(* CODESYS project RoofTrussLibrary.library
   Author: Sawtooth Engineers
   Version: 0.1.0.0
   Description: Containes components and equipment modules for base components of a roof truss core system.
   Title: RoofTrussLibrary
   DefaultNamespace: RTL
   Placeholder: RoofTrussLibrary
   Company: Sawtooth Robotics

Project tree, tasks and I/O mapping:
  libraries: Recipe Management, * (System); SPT Base Types, * (Beckhoff Automation LLC); SPT Components, * (Beckhoff Automation LLC); SPT Event Logger, * (Beckhoff Automation LLC); SPT Motion Control, * (Beckhoff Automation LLC); Tc2_NcDrive, * (Beckhoff Automation GmbH); Tc2_Standard, * (Beckhoff Automation GmbH); Tc2_System, * (Beckhoff Automation GmbH); Tc2_TcpIp, * (Beckhoff Automation GmbH); Tc2_Utilities, * (Beckhoff Automation GmbH); Tc3_Database, * (Beckhoff Automation GmbH); Tc3_EventLogger, * (Beckhoff Automation GmbH); Tc3_JsonXml, * (Beckhoff Automation GmbH); Tc3_PackML_V2, * (Beckhoff Automation GmbH)
  DUTs/
    DB_Logging/
      data type ST_EquipmentModuleLog
    MessageBoxes/
      data type ST_Active_MessageBoxes
      data type ST_MessageBox_Button
      data type ST_MessageBox_Buttons
      data type ST_MessageBox_Data
      data type ST_MessageBox_Messages
      data type ST_MessageBox_Response
    Motion/
      data type E_SpeedOptions
      data type ST_HomingParams
      data type ST_MoveStates
    Recipe/
      data type E_CommandName
      data type E_RamState
      data type ST_AssemblyData
      data type ST_AssemblyEnd
      data type ST_AssemblyStart
      data type ST_AxisRecipe
      data type ST_Board
      data type ST_BoardData
      data type ST_BoardInfo
      data type ST_CSV
      data type ST_CSV_Detail
      data type ST_CSV_Generic
      data type ST_CSV_Line
      data type ST_CSV_Step
      data type ST_Detail_Descriptions
      data type ST_IndexConveyor
      data type ST_KeyValue
      data type ST_PickPlace
      data type ST_PickPlaceDetail
      data type ST_PlateInfo
      data type ST_Plates
      data type ST_PositionInfo
      data type ST_PressRecipe
      data type ST_TrussInfo
    WaitSync/
      data type E_EM_Index
      data type E_WaitSync
      data type ST_WaitSyncManager
    data type E_AssemblyPickState
    data type E_BoardData_Positions
    data type E_CarriageStates
    data type E_Double_Pick_States
    data type E_GrabState
    data type E_Infeed_States
    data type E_Location_IDs
    data type E_MBI_States
    data type E_MoveCarriageState
    data type E_Outfeed_Conveyor_State
    data type E_Outfeed_Conveyor_SubState
    data type E_Press_States
    data type E_ReleaseState
    data type ST_BEPointDefinitions
    data type ST_BoardLengthTest
    data type ST_BoardLengthTestData
    data type ST_ConveyorData
    data type ST_DualChannel_HMIStatus
    data type ST_MGBDoor_HMIStatus
    data type ST_MotorControls_NonStandard
    data type ST_OutfeedConveyorStatus
    data type ST_PackML_Control
    data type ST_PackML_Control_Simplified
    data type ST_RecoveryBoardList
    data type ST_SysConfig
  GVLs/
    global variables Global
  Machine/
    Components/
      BasicSlaveAxis_SOE/
        DUTs/
          HMI/
            data type ST_MyComponent_Command_1
            data type ST_MyComponent_Config_1
            data type ST_MyComponent_HMI_1
            data type ST_MyComponent_Status_1
        Interfaces/
        function block FB_Component_BasicSlaveAxis_SoE [ST]: CyclicLogic, Reset
      Button/
        DUTs/
        Interfaces/
        function block FB_Component_Button [ST]: CyclicLogic, CreateEvents, Initialize, Monitoring, Button_Pressed
      ComponentBase_SR/
        Interfaces/
          interface I_ComponentBase_SR
        function block FB_ComponentBase_SR [ST]: ClearAlarms, RaiseAlarm2Args, Reset
      ControlPendant/
        DUTs/
        Interfaces/
        function block FB_ControlPendant [ST]: CyclicLogic, CreateEvents, Initialize, Monitoring, Mode_Auto, Mode_Idle, Mode_Manual_1, Mode_Manual_2
        function block FB_ControlPendant_Outfeed [ST]: CyclicLogic, CreateEvents, Initialize, Monitoring
      Conveyor/
        DUTs/
          HMI/
        Interfaces/
        function block FB_Conveyor [ST]: CyclicLogic, AlarmRaiseBasic, CreateEvents, Monitoring, SimHoming, ParentResponseDefinitions
      DoubleSolenoidRetractFeedback/
        DUT/
        Interfaces/
        function block FB_DoubleSolenoidRetractFeedback [ST]: Feedback, HardwareInit, RetractedInput
      DualChannelIndicator/
        function block FB_DualChannelMonitor [ST]: CyclicLogic, CreateEvents, Initialize, BothChannelsOK
      Indicator/
        DUTs/
          HMI/
            data type ST_Indicator_Command
            data type ST_Indicator_Config
            data type ST_Indicator_HMI
            data type ST_Indicator_Status
        Interfaces/
          interface I_Indicator: Flash, TurnOff, TurnOn
        function block FB_Component_Indicator [ST]: CyclicLogic, CreateEvents, Flash, Initialize, Monitoring, Reset, TurnOff, TurnOn, Flashing, Off, OffTime, On, OnTime
      IRC5/
        DUTs/
          HMI/
            data type ST_IRC5_Command
            data type ST_IRC5_Config
            data type ST_IRC5_HMI
            data type ST_IRC5_Status
          data type ST_IRC5_Input
          data type ST_IRC5_IO
          data type ST_IRC5_Output
        Interfaces/
          interface I_IRC5
        function block FB_Component_IRC5 [ST]: CyclicLogic, Abort, CreateEvents, EStopReset, Initialize, Monitoring, SignalMapping, Start, Stop, EStopped, InAuto, ParentResponseDefinitions
      MGB_Door/
        DUTs/
          HMI/
        Interfaces/
        function block FB_Component_MGB_Door [ST]: CyclicLogic, HMI_Status, Initialize, AutoStop_CH_OK, Estop_CH_OK, SafetyReset
      Preplate_Rack/
        DUTs/
          HMI/
          data type E_RackState
          data type linked_racks_typ
          data type RackStateMachine
          data type RackStatus
        Interfaces/
        function block FB_Component_Preplate_Rack [ST]: CyclicLogic, Block, Disable, Initialize, IsAvailable, RackLogic, Blocked, InAuto, LinkBlocked
      Robot/
        DUTs/
          data type ST_Robot_Handshake_Input
          data type ST_Robot_Handshake_IO
          data type ST_Robot_Handshake_Output
        Interfaces/
        function block FB_Component_Robot [ST]: CyclicLogic, Clear_DataToSend, CreateEvents, HandshakeSignalMapping, Initialize, Monitoring, PackRecipeData, OtherInputs, OtherOutputs
      Safety/
        DUTs/
          HMI/
        Interfaces/
        function block FB_Component_Safety [ST]: CyclicLogic, CreateEvents, HMI_Indicators, HMI_Status_Estops, HMI_Status_LightCurtains, HMI_Status_Preplate, Initialize, Monitoring, PauseInputs, ResumeInputs, AutostopOK, OutfeedAutostopOK, ParentResponseDefinitions, SafetyOK, SystemState
      StackLight/
        DUTs/
          HMI/
        Interfaces/
          interface I_StackLight: SystemErrorPresent
        function block FB_Component_Stacklight [ST]: CyclicLogic, CreateEvents, Initialize, Monitoring, SystemErrorPresent, SystemState
      StackLight_MBI/
        Interfaces/
          interface I_StackLight_1: MyInput, MyOutput
        function block FB_Component_Stacklight_MBI [ST]: CyclicLogic, CreateEvents, Initialize, Monitoring, MyOutput, SystemErrorPresent
      Template_MyComponent/
        DUTs/
          HMI/
            data type ST_MyComponent_Command
            data type ST_MyComponent_Config
            data type ST_MyComponent_HMI
            data type ST_MyComponent_Status
        Interfaces/
          interface I_MyComponent: SystemErrorPresent, SystemState
        function block FB_Component_MyComponent [ST]: CyclicLogic, CreateEvents, Initialize, Monitoring, MyInput, MyOutput
      VFD/
        DUTs/
          HMI/
        Interfaces/
          interface I_VFD: Jog, Stop
        function block FB_Component_ABB_VFD_EC [ST]: CyclicLogic, Extended, Retracted, Jog, Reset, Stop
        function block FB_Component_ABB_VFD_EIP [ST]: CyclicLogic, Disable, Enable, Initialize, Jog, Monitoring, Reset, Stop, AtSpeed, CommandedVel, Enabled, Faulted, FaultReset, Frequency, FwdActive, JogFwd, JogRvs, ReferenceVel, RvsActive, State, Warning
    EquipmentModules/
      EquipmentModule_SR/
        Interfaces/
          interface I_CommandStepParser: AssemblyEndParse, AssemblyStartParse, BoardInfoParse, BoardParse, NailPlateParse, TrussInfoParse
          interface I_CommandSteps: AssemblyEnd, AssemblyStart, Board, BoardInfo, NailPlate, TrussInfo
          interface I_EquipmentModule_SR: EquipmentModuleID, InSimulation, SafetyOK, SimulationOff, SimulationOn
          interface I_MachineComms: Step, WaitSync
        function block FB_EquipmentModule_SR [ST]: AssemblyEndParse, AssemblyStartParse, BoardInfoParse, BoardParse, IndexConveyorParse, NailPlateParse, PickPlaceParse, TrussInfoParse, CyclicLogic, CyclicLogicSimulation, Step, AssignMessageBox, ComponentMonitor, EM_BufferLogging, HMIControl, LengthFormatString, MotorResetAndEnable, MotorsHome, MotorsInit, MotorsInitAlignGearIn, RaiseAlarm2Args, RaiseMessageBox, RegisterSubmodules, ResetMessageBox, ResetOnResume, RestartStateCheck, SimHoming, SubModuleMonitor, TorqueHoming, TorqueHoming_old, WaitSync_Handler, WaitSync_ReadWrite, WaitSyncCheck, Holding, Resetting, Starting, Suspending, Unholding, Unsuspending, Execute, Idle, Suspended, CurrentStep, EquipmentModuleID, ForceHold, ParentResponseDefinitions, RecoverBoardNum, SafetyOK, TaskState, ClearAlarms, ResetComponents, InSimulation, SimulationOff, SimulationOn
      Functional Layer/
        function block FB_Carriage [ST]: CyclicLogic, Starting, Unholding, Unsuspending, CreateEvents, GrabBoard, HMIControl, Initialize, Monitoring, MotorsInit, MoveIdleOnStarting, ReleaseBoard, SetSpeeds, TestLengthPosCompare, ZPrepMove, ActuatorsClosed, ActuatorsOpen, AxisRef, BoardHeight, BoardSecured, ClearOfBoards, ClearOfCarriages, CloseActuatorsRequest, HoldingBoard, IdlePos, IgnoreSensors, MasterAxis, MoveClearActive, MovementRequested, MoveState, MoveSubState, OpenActuatorsRequest, OverrideSensors, PressPermissions, Request_WS, Response_WS, TargetPos
        function block FB_Handoff [ST]: CyclicLogic, GrabBoard, HMIControl, Initialize, ReleaseBoard, ClampsClosed, ClampsOpen, DisableClamp1, DisableClamp2, HoldingBoard, Location, Request_WS, Response_WS
        function block FB_Infeed [ST]: CyclicLogic, Aborting, Holding, Starting, Stopping, Suspending, ExecuteStep, Execute, Auto, ClearInfeed, CreateEvents, HMIControl, Initialize, Monitoring, ParseBoardData, RoughLengthCheck, SimpAuto, SuperSimpAuto, ActiveInfeedMoving, BoardDataToPass, BoardDropped, BoardReadyForCarriage, Carriage1LengthTesting, Carriage1ResetInfeed_Request, Carriage2_DoublePickCancel_Request, Carriage2ResetInfeed_Request, CarriageClearOfBoardPresentSensor, IgnoreDoublePick, InfeedToInfeedReady, InfeedToInfeedRequest, LineNumber, MoveClearActive, ParentState, ReadyForBoard, Sim_InfeedClear, TestExecute
        function block FB_MBI [ST]: CyclicLogic, Aborting, Holding, Starting, Stopping, Suspending, Unholding, Unsuspending, Aborted, Execute, Held, Idle, Stopped, Suspended, Auto, CreateEvents, HMIControl, Initialize, ManualMode_Forward, ManualMode_Reverse, Monitoring, Production, BoardDropped, LineNumber, MainSafetyOK, ParentState, ReadyForBoard, TestExecute
        function block FB_Outfeed_Jig [ST]: CyclicLogic, Suspending, Unsuspending, ExecuteStep, RunIndexConveyor, RunPickPlace, RunTrussInfo, Aborted, Execute, Held, Idle, Stopped, Suspended, ComponentMonitor, CreateEvents, HMIControl, IndexFull, IndexHalf, Initialize, Monitoring, MotorsInit, NewTrussInfo, OutfeedConveyorLogic, PopulateBoardToArray, AutostopOK, MainSafetyOK, MaxConveyorCount, OutfeedAutostopOK, OutfeedConveyorStatus, ParentState, PickPlace_Done_ENUM, PickPlace_Ready_ENUM
        function block FB_Preplate [ST]: CyclicLogic, Execute, HMIControl, Initialize, InAuto
        function block FB_Press [ST]: CyclicLogic, Aborting, Clearing, Holding, Starting, Stopping, Suspending, Unholding, Unsuspending, AssemblyEnd, AssemblyStart, ExecuteDetail, ExecuteStep, Execute, DoublePickNailPlatePosCheck, HMIControl, Initialize, MotorsInit, PressLogic, BoardDataToPass, DoublePickData_Ready, DoublePickData_Sent, DoublePickDataToPass, NailplateCountData_Ready, NailplateCountData_Sent, NailplateDataToPass, PressRobotPermissionToEnter
        function block FB_Robot [ST]: CyclicLogic, CyclicLogicSimulation, Aborting, Clearing, Completing, Holding, Resetting, Starting, Stopping, Suspending, Unholding, Unsuspending, NailPlate, Execute, ExtractNumFromString, HMIControl, Initialize, WaitSync_Robot, DryRun, OtherInputs, OtherOutputs, SubModuleMonitor
        function block FB_Robot_Outfeed [ST]: CyclicLogic, CyclicLogicSimulation, ExecuteDetail, ExecuteDetail_SIM, ExecuteStep, HMIControl, Initialize, UI_MessageBox, PickPlaceDataToPass
        function block FB_Robot_PrePlate [ST]: CyclicLogic, CyclicLogicSimulation, ExecuteDetail, ExecuteDetail_SIM, ExecuteStep, HMIControl, Initialize, UI_MessageBox
        function block FB_Robot_Press [ST]: CyclicLogic, CyclicLogicSimulation, ExecuteDetail, ExecuteDetail_SIM, ExecuteStep, HMIControl, Initialize, UI_MessageBox
      Info Layer/
        function block _FB_EquipmentModule_Info [ST]: CyclicLogic, Aborting, FindBoardForRecovery, Task
      SamComm/
        DUTs/
          HMI/
          data type E_ContentType
          data type E_MessageCategory
          data type E_MessageStatus
          data type E_SAMCommStateMachine
          data type E_TaskState
          data type ST_Alert
          data type ST_Message
          data type ST_Messages
          data type ST_PLC
          data type ST_RFT
          data type ST_Status
          data type ST_Task
          data type ST_Task_Info
          data type ST_TaskREF
          data type ST_TaskStatus
        Helper POUs/
          function block FB_FrameFifo [ST]: AddTail, Clear, RemoveHead, Send
          function block FB_LogFifo [ST]: Clear, Error, Message, Remove
        function block FB_ClientConnection [ST]
        function block FB_SamComm [ST]: CyclicLogic, CheckForRFT, CheckForStatusUpdate, ComposeRequestForInfo, ComposeRFT, ComposeStatus, ExtractMetaData, GenUUID, InfeedLineNumberCheck, IsIdleTask, ParseCSVData, ProcessReceivedMessage, STRING_TO_E_CommandName, Application, CreateEvents, Initialize, RaiseAlarm2Args, OutfeedConveyorStatus_Jig2, OutfeedConveyorStatus_Jig3, Tasks
      Templates/
    Events/
      AMDTruss.tmc
    FunctionBlocks/
      Occupy Press Street/
        data type E_GateKeeperState
        data type ST_MediatorInterface
      PulseGenerator/
        Interfaces/
          interface I_PulseGenerator: OffTime, OnTime, PulseOutput
        function block FB_PulseGenerator [ST]: CyclicLogic, OffTime, OnTime, PulseOutput
    HMI Connections/
      function block FB_ControlSource_HMI [ST]: CyclicLogic, Control, ModeChanged, StateChanged, ForceHoldRequested, Initialize, Registered
      function block FB_ControlSource_HMI_Machine [ST]: CyclicLogic
      function block FB_ControlSource_MBI [ST]: CyclicLogic, Control, ModeChanged, StateChanged, Initialize, Registered
  00000000-0000-0000-0000-000000000000|Machine\Events\AMDTruss.tmc
  Project Information/
    function F_GetCompany [ST]
    function F_GetTitle [ST]
    function F_GetVersion [ST]
  Version/
    global variables Global_Version
  text list GlobalTextList
*)

// DUTs/DB_Logging/ST_EquipmentModuleLog
TYPE
    ST_EquipmentModuleLog : STRUCT
        Timestamp   : DT;
        ModuleName  : STRING(32);
        PackMLState : STRING(32);
        Message     : STRING(255);
    END_STRUCT
END_TYPE

// DUTs/MessageBoxes/ST_Active_MessageBoxes
TYPE
    ST_Active_MessageBoxes : STRUCT
        SelectedTabIndex          : USINT;
        MessageBox_Data           : ARRAY[1..30] OF ST_MessageBox_Data;
        Displayed_MessageBox_Data : ST_MessageBox_Data;
        ErrorSolution             : USINT;
        ErrorAcknowledge          : BOOL;
    END_STRUCT
END_TYPE

// DUTs/MessageBoxes/ST_MessageBox_Button
TYPE
    ST_MessageBox_Button : STRUCT
        Text    : STRING;
        Visible : BOOL;
    END_STRUCT
END_TYPE

// DUTs/MessageBoxes/ST_MessageBox_Buttons
TYPE
    ST_MessageBox_Buttons : STRUCT
        Button1 : ST_MessageBox_Button;
        Button2 : ST_MessageBox_Button;
        Button3 : ST_MessageBox_Button;
        Button4 : ST_MessageBox_Button;
        Button5 : ST_MessageBox_Button;
    END_STRUCT
END_TYPE

// DUTs/MessageBoxes/ST_MessageBox_Data
TYPE
    ST_MessageBox_Data : STRUCT
        Equipment_Module        : E_EM_Index;
        Equipment_Module_String : STRING;
        TimeStamp               : STRING;
        Header                  : STRING[80];
        Icon                    : USINT;
        Severity                : TcEventSeverity;
        Messages                : ST_MessageBox_Messages;
        Buttons                 : ST_MessageBox_Buttons;
        ErrorPresent            : BOOL;
        ErrorNumber             : UINT;
    END_STRUCT
END_TYPE

// DUTs/MessageBoxes/ST_MessageBox_Messages
TYPE
    ST_MessageBox_Messages : STRUCT
        Message1 : STRING[80];
        Message2 : STRING[80];
        Message3 : STRING[80];
        Message4 : STRING[80];
        Message5 : STRING[80];
        Message6 : STRING[80];
        Message7 : STRING[80];
    END_STRUCT
END_TYPE

// DUTs/MessageBoxes/ST_MessageBox_Response
TYPE
    ST_MessageBox_Response : STRUCT
        ErrorRaised      : BOOL;
        ErrorAcknowledge : BOOL;
        ErrorSolution    : USINT;
    END_STRUCT
END_TYPE

// DUTs/Motion/E_SpeedOptions
{attribute 'qualified_only'}
{attribute 'strict'}
{attribute 'to_string'}
TYPE
    E_SpeedOptions : (
        AUTO        := 1,
        MANUAL      := 2,
        MAINTENANCE := 3,
        TESTING1    := 4,
        TESTING2    := 5,
        TESTING3    := 6,
        TESTING4    := 7,
        TESTING5    := 8
    );
END_TYPE

// DUTs/Motion/ST_HomingParams
TYPE
    ST_HomingParams : STRUCT
        ReadParams               : SPT_Motion_Control.MC_ReadParameter;
        WriteNegLim              : SPT_Motion_Control.MC_WriteBoolParameter;
        WritePosLim              : SPT_Motion_Control.MC_WriteBoolParameter;
        AxisParams               : SPT_Motion_Control.MC_AxisParameter;
        SetPositionHomingRoutine : FB_HomeRoutine_SetPosition;
        TorqueControl            : SPT_Motion_Control.MC_TorqueControl;
        TorqueControlParams      : SPT_Motion_Control.ST_TorqueControlOptions;
        HardStopHomingRoutine    : FB_HomeRoutine_HardStop;
        HardStopHomingParams     : ST_StepBlockLagBasedParameters;
        SetPositionOffset        : SPT_Motion_Control.FB_CoEAX8000SetPositionOffset;
        HomingTON                : TON;
        Execute_WriteLimit       : BOOL;
        EnablePosLim             : BOOL;
        EnableNegLim             : BOOL;
        HomingState              : DINT;
        HomePosMax               : LREAL;
        HomePosMin               : LREAL;
    END_STRUCT
END_TYPE

// DUTs/Motion/ST_MoveStates
TYPE
    ST_MoveStates : STRUCT
        Idle    : UDINT;
        Pick    : UDINT;
        Hold    : UDINT;
        Clear   : UDINT;
        Drop    : UDINT;
        Grab    : UDINT;
        Release : UDINT;
    END_STRUCT
END_TYPE

// DUTs/Recipe/E_CommandName
{attribute 'qualified_only'}
{attribute 'strict'}
{attribute 'to_string'}
TYPE
    E_CommandName : (
        Unknown       := 0,
        AssemblyStart := 1,
        TrussInfo     := 2,
        PuckMove      := 3,
        PickPlace     := 4,
        IndexConveyor := 5,
        ManualBoard   := 6,
        BoardInfo     := 7,
        Board         := 8,
        NailPlate     := 9,
        ManualPlate   := 10,
        AssemblyEnd   := 11
    );
END_TYPE

// DUTs/Recipe/E_RamState
{attribute 'qualified_only'}
{attribute 'strict'}
{attribute 'to_string'}
TYPE
    E_RamState : (
        rsINIT,
        rsIDLE,
        rsFULL_RETRACT,
        rsFULL_EXTEND,
        rsSEND_TO_POSITION,
        rsEXTEND_TO_BACKER,
        rsEXTEND_TO_CLOSED_PREP,
        rsEXTEND_TO_CLOSED,
        rsFAILED_TO_CYCLE,
        rsEXTENDING_TO_PRESSURE,
        rsEXTEND_TO_PRESSURE,
        rsRETRACT_FOR_INDEX,
        rsUNDEFINED,
        rsERROR
    );
END_TYPE

// DUTs/Recipe/ST_AssemblyData
TYPE
    ST_AssemblyData : STRUCT
        Boards : ARRAY[1..MAX_NUMBER_OF_BOARDS] OF ST_BoardData;
    END_STRUCT
END_TYPE

// DUTs/Recipe/ST_AssemblyEnd
TYPE
    ST_AssemblyEnd : STRUCT
        SeqID : UDINT;
    END_STRUCT
END_TYPE

// DUTs/Recipe/ST_AssemblyStart
TYPE
    ST_AssemblyStart : STRUCT
        ComponentID : T_MaxString;
    END_STRUCT
END_TYPE

// DUTs/Recipe/ST_AxisRecipe
TYPE
    ST_AxisRecipe : STRUCT
        Velocity     : LREAL := 150;
        Acceleration : LREAL := 300;
        Torque       : LREAL := 100;
    END_STRUCT
END_TYPE

// DUTs/Recipe/ST_Board
TYPE
    ST_Board : STRUCT
        BoardID                 : STRING;
        BoardWidth              : REAL;
        BoardHeight             : REAL;
        BoardLength             : REAL;
        BoardNumber             : INT;
        LeadingEdgeBevelOffset  : REAL;
        TrailingEdgeBevelOffset : REAL;
    END_STRUCT
END_TYPE

// DUTs/Recipe/ST_BoardData
TYPE
    ST_BoardData : STRUCT
        BoardID                       : STRING;
        BoardWidth                    : REAL;
        BoardHeight                   : REAL;
        BoardLength                   : REAL;
        BoardLength_Measured          : BOOL;
        BoardNumber                   : INT;
        Plates_Total                  : UDINT;
        Plates_Placed                 : UDINT;
        TotalPlateCount_Data_Received : BOOL;
        LeadingEdgeBevelOffset        : REAL;
        TrailingEdgeBevelOffset       : REAL;
        PickOffset                    : REAL;
        DoublePickNeeded              : BOOL;
        DoublePickVerified            : BOOL;
        DoublePicked                  : BOOL;
        IgnoreSensors                 : BOOL;
        FrontEdgePos                  : REAL;
        BackEdgePos                   : REAL;
        LocationStr                   : STRING;
        LengthFormatted_str           : STRING;
        Positions                     : ARRAY[1..MAX_NUMBER_OF_POSITIONS] OF ST_PositionInfo;
        Plates                        : ARRAY[1..MAX_NUMBER_OF_PLATES] OF ST_PlateInfo;
        PickPlaceInfo                 : ST_PickPlaceDetail; // Pick and Place Data Specific to Outfeed
        ConveyorIndexInfo             : INT; // Conveyor Index data for Outfeed
    END_STRUCT
END_TYPE

// DUTs/Recipe/ST_BoardInfo
TYPE
    ST_BoardInfo : STRUCT
        BoardID     : STRING;
        BoardWidth  : REAL;
        BoardHeight : REAL;
        BoardLength : REAL;
        BoardNumber : INT;
        TotalPlates : INT;
    END_STRUCT
END_TYPE

// DUTs/Recipe/ST_CSV
TYPE
    ST_CSV : STRUCT
        Steps : ARRAY[1..MAX_STEP_COUNT] OF ST_CSV_Step;
    END_STRUCT
END_TYPE

// DUTs/Recipe/ST_CSV_Detail
TYPE
    ST_CSV_Detail : STRUCT
        DetailID  : UDINT;
        DataCount : UDINT;
        Datas     : ARRAY[1..MAX_DATA_COUNT] OF T_MaxString;
    END_STRUCT
END_TYPE

// DUTs/Recipe/ST_CSV_Generic
TYPE
    ST_CSV_Generic : STRUCT
        CSVLines : ARRAY[1..600] OF ST_CSV_Line;
    END_STRUCT
END_TYPE

// DUTs/Recipe/ST_CSV_Line
TYPE
    ST_CSV_Line : STRUCT
        Fields : ARRAY[1..MAX_DATA_COUNT] OF T_MaxString;
    END_STRUCT
END_TYPE

// DUTs/Recipe/ST_CSV_Step
TYPE
    ST_CSV_Step : STRUCT
        seqName     : E_CommandName;
        seqID       : UDINT;
        DetailCount : UDINT;
        Details     : ARRAY[1..MAX_DETAIL_COUNT] OF ST_CSV_Detail;
    END_STRUCT
END_TYPE

// DUTs/Recipe/ST_Detail_Descriptions
TYPE
    ST_Detail_Descriptions : STRUCT
        Detail_Key : ARRAY[1..Global.MAX_DETAIL_COUNT] OF ST_KeyValue;
    END_STRUCT
END_TYPE

// DUTs/Recipe/ST_IndexConveyor
TYPE
    ST_IndexConveyor : STRUCT
        ConvIndex : INT;
    END_STRUCT
END_TYPE

// DUTs/Recipe/ST_KeyValue
TYPE
    ST_KeyValue : STRUCT
        ID  : STRING;
        Typ : STRING;
    END_STRUCT
END_TYPE

// DUTs/Recipe/ST_PickPlace
TYPE
    ST_PickPlace : STRUCT
        ID        : STRING;
        Width     : REAL;
        Height    : REAL;
        Length    : REAL;
        Number    : INT;
        boardType : STRING;
        XPos      : REAL;
        YPos      : REAL;
        ZPos      : REAL;
        ZRot      : REAL;
        ConvIndex : INT;
    END_STRUCT
END_TYPE

// DUTs/Recipe/ST_PickPlaceDetail
TYPE
    ST_PickPlaceDetail : STRUCT
        MemberType : STRING;
        XPos       : REAL;
        YPos       : REAL;
        ZPos       : REAL;
        ZRot       : REAL;
        ConvIndex  : INT;
    END_STRUCT
END_TYPE

// DUTs/Recipe/ST_PlateInfo
TYPE
    ST_PlateInfo : STRUCT
        BoardID         : STRING;
        PlateID         : STRING;
        PlateNumber     : INT;
        PlateDimensions : STRING; // Dimension information of the plate (length, width, gauge)
        PlateGauge      : STRING;
        PlateWidth      : REAL;
        PlateHeight     : REAL;
        PlatePlaceX     : REAL;
        PlatePlaceY     : REAL;
        PlatePlaceAngle : REAL;
        TopOrBottom     : STRING; // Indicates if plate is on top or bottom of the board
    END_STRUCT
END_TYPE

// DUTs/Recipe/ST_Plates
TYPE
    ST_Plates : STRUCT
        Plates : ARRAY[1..MAX_NUMBER_OF_PLATES] OF ST_PlateInfo;
    END_STRUCT
END_TYPE

// DUTs/Recipe/ST_PositionInfo
TYPE
    ST_PositionInfo : STRUCT
        Position     : REAL;
        PositionType : INT;
    END_STRUCT
END_TYPE

// DUTs/Recipe/ST_PressRecipe
TYPE
    ST_PressRecipe : STRUCT
        State               : E_RamState;
        State_Previous      : E_RamState;
        State_Response      : E_RamState;
        State_Str           : STRING;
        State_Previous_Str  : STRING;
        State_Response_Str  : STRING;
        PressOnRetract      : BOOL;
        Pressure            : UINT;
        SubState            : UINT;
        OpenPosition        : UINT := 70;
        BackerPosition      : UINT := 163;
        ClosedPosition      : UINT := 170;
        AtTop               : BOOL;
        AtWork              : BOOL;
        Axis                : ST_AxisRecipe;
        TorqueOptions       : SPT_Motion_Control.ST_TorqueControlOptions;
        TorqueControl       : SPT_Motion_Control.MC_TorqueControl;
        DriveOpMode_Read    : SPT_Motion_Control.MC_ReadDriveOperationMode;
        DriveOpMode_Write   : SPT_Motion_Control.MC_ReadDriveOperationMode;
        DriveOpMode_Options : SPT_Motion_Control.ST_DriveOperationModeOptions;
        Execute_TorqueMove  : BOOL;
    END_STRUCT
END_TYPE

// DUTs/Recipe/ST_TrussInfo
TYPE
    ST_TrussInfo : STRUCT
        TrussID          : STRING;
        MemberCount      : INT;
        TrussXOffs       : REAL;
        TrussYOffs       : REAL;
        TrussLength      : REAL;
        TrussWidth       : REAL;
        PressBeforeTruss : BOOL;
        LeftEndType      : STRING; // Type of the left end (specific to Outfeed)
        RightEndType     : STRING; // Type of the right end (specific to Outfeed)
    END_STRUCT
END_TYPE

// DUTs/WaitSync/E_EM_Index
{attribute 'qualified_only'}
{attribute 'strict'}
{attribute 'to_string'}
TYPE
    E_EM_Index : (
        EMPTY          := 0,
        MBI_1          := 1,
        MBI_2          := 2,
        INFEED_1       := 3,
        INFEED_2       := 4,
        CARRIAGE_1     := 5,
        CARRIAGE_2     := 6,
        CARRIAGE_3     := 7,
        HANDOFF_1      := 8,
        HANDOFF_2      := 9,
        HANDOFF_3      := 10,
        HANDOFF_4      := 11,
        PICK_1         := 12,
        PICK_2         := 13,
        PICK_3         := 14,
        PICK_4         := 15,
        PRESS          := 16,
        PRESS_ROBOT    := 17,
        PREPLATE_CELL  := 18,
        PREPLATE_ROBOT := 19,
        OUTFEED_ROBOT  := 20,
        OUTFEED_JIG2   := 21,
        OUTFEED_JIG3   := 22,
        AMD_TASK       := 23,
        INFEED_TASK    := 24,
        PREPLATE_TASK  := 25,
        PRESS_TASK     := 26,
        TRANSPORTER    := 27,
        SAMCOMMS       := 28,
        MACHINE        := 29
    );
END_TYPE

// DUTs/WaitSync/E_WaitSync
{attribute 'qualified_only'}
{attribute 'strict'}
{attribute 'to_string'}
TYPE
    E_WaitSync : (
        EMPTY                                := 0,
        BOARD_READY_FOR_NAILPLATE            := 1,
        CARRIAGE1_INFEED_DATA_CONFIRMED      := 2,
        CARRIAGE1_INFEED_BOARD_READY         := 3,
        CARRIAGE1_INFEED_BOARD_PICKED        := 4,
        CARRIAGE2_INFEED_DOUBLE_PICK_REQUEST := 5,
        CARRIAGE2_INFEED_DOUBLE_PICK_READY   := 6,
        HANDOFF2_PRESS_TOTAL_NP_COUNT        := 7,
        HANDOFF2_PRESS_DOUBLE_PICK           := 8,
        CARRIAGE2_PRESS_READY_FOR_BOARD      := 9,
        CARRIAGE2_PRESS_NAILPLATE_DONE       := 10,
        CARRIAGE2_PRESS_BOARD_IN_POSITION    := 11,
        CARRIAGE2_CARRIAGE1_GEARED_IN        := 12,
        CARRIAGE2_CARRIAGE1_GEAR_IN          := 13,
        CARRIAGE2_CARRIAGE1_GEAR_OUT         := 14,
        CARRIAGE1_INFEED_BOARD_PICKING       := 15,
        CARRIAGE2_INFEED_DOUBLE_PICK_DONE    := 16,
        CARRIAGE1_INFEED_PICKING             := 17,
        CARRIAGE1_INFEED_BOARD_LENGTH_CHECK  := 18,
        CARRIAGE2_INFEED_BOARD_LENGTH_CHECK  := 19,
        INFEED1_MBI_DROP_BOARD               := 20,
        INFEED1_INFEED2_RELEASE_BOARD        := 21,
        INFEED2_MBI_DROP_BOARD               := 22,
        NAILPLATE_READY_TO_PLACE             := 50,
        NAILPLATE_PLACED                     := 51,
        PRESS_ROBOT_PERMISSION_GRANTED       := 52,
        PRESS_PREPLATE_SIM_SYNC              := 53,
        PICK1_ASSEMBLY_BOARD_READY           := 70,
        PICK1_ASSEMBLY_OPEN_GRIPPERS         := 71,
        PICK1_ASSEMBLY_BOARD_CLEAR           := 72,
        PICK1_ASSEMBLY_PICKING_BOARD         := 73,
        OUTFEED_JIG2_PICKPLACE_READY         := 74,
        OUTFEED_JIG2_PICKPLACE_DONE          := 75,
        OUTFEED_JIG3_PICKPLACE_READY         := 76,
        OUTFEED_JIG3_PICKPLACE_DONE          := 77
    );
END_TYPE

// DUTs/WaitSync/ST_WaitSyncManager
TYPE
    ST_WaitSyncManager : STRUCT
        ID         : E_WaitSync;
        Active     : BOOL;
        AreaNeeded : ARRAY[1..30] OF BOOL;
        State      : UDINT;
    END_STRUCT
END_TYPE

// DUTs/E_AssemblyPickState
{attribute 'strict'}
{attribute 'to_string'}
TYPE
    E_AssemblyPickState : (
        BOARD_READY_WS        := 0,
        OPEN_GRIPPERS_WS      := 20,
        OPEN_GRIPPERS         := 30,
        PICKING_BOARD_WS      := 35,
        BOARD_CLEAR_WS        := 40,
        PICK_DONE             := 50,
        SIM_JIG2READYPLACE_WS := 200,
        SIM_JIG2PLACEDONE_WS  := 201,
        SIM_JIG3READYPLACE_WS := 202,
        SIM_JIG3PLACEDONE_WS  := 203,
        PICK_ERROR            := 999
    );
END_TYPE

// DUTs/E_BoardData_Positions
{attribute 'qualified_only'}
{attribute 'strict'}
{attribute 'to_string'}
TYPE
    E_BoardData_Positions : (
        INVALID                  := 0,
        CARRIAGE_1INFEED_HANDOFF := 1,
        CARRIAGE_12_HANDOFF      := 2,
        CARRIAGE_23_HANDOFF      := 3,
        BOARD_DROP               := 4,
        GEAR_IN_SYNC             := 5
    );
END_TYPE

// DUTs/E_CarriageStates
{attribute 'qualified_only'}
{attribute 'strict'}
{attribute 'to_string'}
TYPE
    E_CarriageStates : (
        IDLE                              := 0,
        HOLDING_BOARD                     := 1,
        PICK                              := 2,
        PICK_CONFIRM                      := 3,
        PRESS_READY_FOR_BOARD             := 4,
        PRESS_BOARD_IN_PLACE              := 5,
        PRESS_BOARD_CLEAR_CHECK           := 6,
        PRESS_NAILPLATE_DONE              := 7,
        PRESS_NAILPLATE_DONE_CHECK        := 8,
        NAILPLATE_DATA_CONFIRMATION       := 9,
        PRESS_BOARD_CLEAR                 := 10,
        DROPPING                          := 11,
        DROP                              := 12,
        DROP_CONFIRM                      := 13,
        HOLD_BOARD_FOR_PICK               := 14,
        GEAR_IN_MOVE                      := 15,
        GEAR_IN_WAIT                      := 16,
        GEARED_IN                         := 17,
        NAILPLATE_POS_CALCULATION         := 18,
        GEAR_OUT_WAIT                     := 19,
        GEAR_OUT_HS                       := 20,
        PRESS_MOVE_BOARD_TO_POSITION      := 21,
        PICKING                           := 22,
        MOVE_PREP                         := 23,
        LENGTH_CHECK                      := 24,
        CARRIAGE_RESUME_AFTER_WRONG_BOARD := 25,
        RESET                             := 99
    );
END_TYPE

// DUTs/E_Double_Pick_States
{attribute 'strict'}
{attribute 'to_string'}
TYPE
    E_Double_Pick_States : (
        DP_REQUEST_WS    := 0,
        DP_SECURE        := 10,
        DP_PICK_READY_WS := 20,
        DP_RETRACT_CLAMP := 30,
        DP_PICK_DONE_WS  := 40,
        DP_GEAR_IN_WS    := 50,
        DP_GEAR_IN       := 60,
        DP_GEARED_IN_WS  := 70,
        DP_ERROR         := 999
    );
END_TYPE

// DUTs/E_GrabState
{attribute 'strict'}
{attribute 'to_string'}
TYPE
    E_GrabState : (
        GRAB_START        := 0,
        GRAB_MOVE_CHECK   := 10,
        GRAB_TORQUE       := 20,
        GRAB_FINISHED     := 40,
        GRAB_VERIFY       := 50,
        GRAB_RESUME_START := 60,
        GRAB_ERROR        := 999
    );
END_TYPE

// DUTs/E_Infeed_States
{attribute 'strict'}
{attribute 'to_string'}
TYPE
    E_Infeed_States : (
        INF_IDLE                    := 0,
        INF_CONVEY                  := 10,
        INF_BOARD_FOUND             := 20,
        INF_BOARD_CHECK             := 30,
        INF_ROUGH_LENGTH_CHECK      := 35,
        INF_BOARD_READY             := 40,
        INF_BOARD_READY_WS          := 50,
        INF_BOARD_PICKING_WS        := 55,
        INF_RETRACT_CLAMPS          := 60,
        INF_BOARD_PICKED_WS         := 90,
        INF_BOARD_LENGTH_CHECK_CAR1 := 95,
        INF_BOARD_LENGTH_CHECK_CAR2 := 96,
        INF_DOUBLE_PICK             := 100,
        INF_WRONG_BOARD             := 200,
        INF_ERROR                   := 999
    );
END_TYPE

// DUTs/E_Location_IDs
{attribute 'qualified_only'}
{attribute 'strict'}
{attribute 'to_string'}
TYPE
    E_Location_IDs : (
        INVALID        := 0,
        CARRIAGE_1     := 1,
        CARRIAGE_2     := 2,
        CARRIAGE_3     := 3,
        INFEED         := 4,
        PRE_PRESS      := 5,
        POST_PRESS     := 6,
        ASSEM_HANDOFF  := 7,
        PICK_1_HANDOFF := 8,
        PICK_1         := 9
    );
END_TYPE

// DUTs/E_MBI_States
{attribute 'strict'}
{attribute 'to_string'}
TYPE
    E_MBI_States : (
        acIDLE                := 0,
        acINDEX_FORWARD       := 1,
        acINDEX_TO_DOG_SENSOR := 2,
        acWAIT_INFEED_READY   := 3,
        acDUMP_BOARD          := 4,
        acTOP_SPOT_POPULATED  := 5,
        acBOARD_LOST          := 6,
        acSTOP                := 7,
        acWAIT_READY          := 8,
        FORWARD               := 9,
        acERROR               := 999
    );
END_TYPE

// DUTs/E_MoveCarriageState
{attribute 'strict'}
{attribute 'to_string'}
TYPE
    E_MoveCarriageState : (
        INIT                   := 0,
        MOVEMENT_CHECK         := 10,
        GRAB_AFTER_MOVE        := 20,
        SECURE_AFTER_MOVE      := 30,
        RELEASE_AFTER_MOVE     := 40,
        CARRIAGE_CHECK_MESSAGE := 50,
        SENSOR_CHECK_MESSAGE   := 60,
        REENABLE_RESUME_MOVE   := 70,
        DONE                   := 100
    );
END_TYPE

// DUTs/E_Outfeed_Conveyor_State
{attribute 'qualified_only'}
{attribute 'strict'}
{attribute 'to_string'}
TYPE
    E_Outfeed_Conveyor_State : (
        INVALID           := 0,
        IDLE              := 1,
        INDEX_PREP        := 2,
        INDEXING          := 3,
        INDEX_HALF_PREP   := 4,
        INDEXING_HALF     := 5,
        RECEIVE_PREP      := 6,
        RECEIVING         := 7,
        OCCUPIED          := 8,
        RESET             := 9,
        BUILD_IN_PROGRESS := 10,
        AUTO_RETRACT      := 20,
        ERROR             := 999
    );
END_TYPE

// DUTs/E_Outfeed_Conveyor_SubState
{attribute 'strict'}
{attribute 'to_string'}
TYPE
    E_Outfeed_Conveyor_SubState : (
        CONV_MOVE_ASSIGN       := 0,
        CONV_MOVE_DONE_CHECK   := 10,
        CONV_DATA_CONFIRMATION := 20,
        CONV_RESET_MOTOR       := 30,
        CONV_ERROR             := 999
    );
END_TYPE

// DUTs/E_Press_States
{attribute 'strict'}
{attribute 'to_string'}
TYPE
    E_Press_States : (
        PRESS_INIT                  := 0,
        NP_READY_TO_PLACE_WS        := 10,
        ROBOT_PERMISSION_REQUEST    := 11,
        ROBOT_PERMISSION_GRANTED_WS := 15,
        NP_PLACED_WS                := 20,
        NP_PREP_POS                 := 25,
        READY_FOR_BOARD_WS          := 30,
        BOARD_IN_POSITION_WS        := 35,
        PRESSING_NAILPLATE          := 40,
        RETRACTING_FOR_INDEX        := 41,
        NP_DONE_WS                  := 50
    );
END_TYPE

// DUTs/E_ReleaseState
{attribute 'strict'}
{attribute 'to_string'}
TYPE
    E_ReleaseState : (
        RELEASE_START      := 0,
        RELEASE_MOVE       := 10,
        RELEASE_MOVE_CHECK := 20,
        RELEASE_FINISHED   := 30,
        RELEASE_ERROR      := 999
    );
END_TYPE

// DUTs/ST_BEPointDefinitions
TYPE
    ST_BEPointDefinitions : STRUCT
        MinCarriagePos  : REAL;
        Infeed          : REAL;
        PrePress        : REAL;
        PostPress       : REAL;
        AssemblyHandoff : REAL;
        PickPoint_1     : REAL;
        MaxCarriagePos  : REAL;
    END_STRUCT
END_TYPE

// DUTs/ST_BoardLengthTest
TYPE
    ST_BoardLengthTest : STRUCT
        LengthCalculated : ARRAY[1..10] OF LREAL;
    END_STRUCT
END_TYPE

// DUTs/ST_BoardLengthTestData
TYPE
    ST_BoardLengthTestData : STRUCT
        VelocityArray : ARRAY[1..10] OF ST_BoardLengthTest;
    END_STRUCT
END_TYPE

// DUTs/ST_ConveyorData
TYPE
    ST_ConveyorData : STRUCT
        ConveyorID       : STRING;
        ConveyorStateStr : STRING;
        TargetPos        : LREAL;
        State            : E_Outfeed_Conveyor_State := E_Outfeed_Conveyor_State.IDLE;
        TrussInfo        : ST_TrussInfo;
        CurrentTruss     : STRING;
        BoardsPresent    : ARRAY[1..50] OF ST_PickPlace;

        ActualPosition : LREAL;

        ReadyToIndexHalf      : BOOL;
        HalfIndexCompleted    : BOOL;
        SubState              : E_Outfeed_Conveyor_SubState := E_Outfeed_Conveyor_SubState.CONV_MOVE_ASSIGN;
        ConveyorLength        : LREAL                       := 7075; //mm
        ReadyToIndex          : BOOL                        := FALSE;
        ReadyToOutfeed        : BOOL                        := FALSE;
        ReadyToReceive        : BOOL                        := FALSE;
        ReadyForSlideOut      : BOOL                        := FALSE;
        ClearConveyor         : BOOL                        := FALSE;
        ConveyorVelocity      : INT                         := 500;
        ManualControlSelected : BOOL                        := FALSE;
    END_STRUCT
END_TYPE

// DUTs/ST_DualChannel_HMIStatus
TYPE
    ST_DualChannel_HMIStatus : STRUCT
		Name : STRING;
		Status_Usint : USINT;
		Status_Str : STRING;		
    END_STRUCT
END_TYPE

// DUTs/ST_MGBDoor_HMIStatus
TYPE
    ST_MGBDoor_HMIStatus : STRUCT
		DoorName : STRING;
		AutoStopStatus_Usint : USINT;
		AutoStopStatus_Str : STRING;
		EStopStatus_Usint : USINT;
		EStopStatus_Str : STRING;		
    END_STRUCT
END_TYPE

// DUTs/ST_MotorControls_NonStandard
TYPE
    ST_MotorControls_NonStandard : STRUCT
        MotorCmd     : ARRAY[1..10] OF BOOL;
        Temp_R_Trig : ARRAY[1..10] OF R_TRIG;
    END_STRUCT
END_TYPE

// DUTs/ST_OutfeedConveyorStatus
TYPE
    ST_OutfeedConveyorStatus : STRUCT
        Occupied : USINT;
        Total    : UDINT;
    END_STRUCT
END_TYPE

// DUTs/ST_PackML_Control
TYPE
    ST_PackML_Control : STRUCT
        CurrentMode  : E_PMLUnitMode;
        ModeCommand  : E_PMLUnitMode;
        CurrentState : E_PMLState;
        StateCommand : E_PMLCommand;
        ModeNames    : ARRAY[0..31] OF STRING;
    END_STRUCT
END_TYPE

// DUTs/ST_PackML_Control_Simplified
TYPE
    ST_PackML_Control_Simplified : STRUCT
        AbortPermissive     : BOOL;
        HoldPermissive      : BOOL;
        ResetPermissive     : BOOL;
        StartPermissive     : BOOL;
        StopPermissive      : BOOL;
        AbortPressed        : BOOL;
        HoldPressed         : BOOL;
        ResetPressed AT %I* : BOOL;
        StartPressed AT %I* : BOOL;
        StopPressed  AT %I* : BOOL;
    END_STRUCT
END_TYPE

// DUTs/ST_RecoveryBoardList
TYPE
    ST_RecoveryBoardList : STRUCT
        BoardID : STRING;
        Index   : STRING;
        Length  : STRING;
    END_STRUCT
END_TYPE

// DUTs/ST_SysConfig
TYPE
    ST_SysConfig : STRUCT
        TableLength_mm  : LREAL;
        FastHandshakes  : BOOL;
        VersionNumber   : USINT;
        HardwareVersion : USINT;
        OutfeedType     : STRING;
        PressInterface  : INT;
        UsedCarriages   : USINT;
    END_STRUCT
END_TYPE

// Machine/Components/BasicSlaveAxis_SOE/DUTs/HMI/ST_MyComponent_Command_1
TYPE
    ST_MyComponent_Command_1 : STRUCT
        Extend  : BOOL;
        Retract : BOOL;
    END_STRUCT
END_TYPE

// Machine/Components/BasicSlaveAxis_SOE/DUTs/HMI/ST_MyComponent_Config_1
TYPE
    ST_MyComponent_Config_1 : STRUCT
        ExtendTime  : LREAL;
        RetractTime : LREAL;
    END_STRUCT
END_TYPE

// Machine/Components/BasicSlaveAxis_SOE/DUTs/HMI/ST_MyComponent_HMI_1
TYPE
    ST_MyComponent_HMI_1 : STRUCT
        Config  : ST_MyComponent_Config;
        Command : ST_MyComponent_Command;
        Status  : ST_MyComponent_Status;
    END_STRUCT
END_TYPE

// Machine/Components/BasicSlaveAxis_SOE/DUTs/HMI/ST_MyComponent_Status_1
TYPE
    ST_MyComponent_Status_1 : STRUCT
        Extended   : BOOL;
        Retracted  : BOOL;
        Extending  : BOOL;
        Retracting : BOOL;
    END_STRUCT
END_TYPE

// Machine/Components/Indicator/DUTs/HMI/ST_Indicator_Command
TYPE
    ST_Indicator_Command : STRUCT
        TurnOn  : BOOL;
        TurnOff : BOOL;
        Flash   : BOOL;
    END_STRUCT
END_TYPE

// Machine/Components/Indicator/DUTs/HMI/ST_Indicator_Config
TYPE
    ST_Indicator_Config : STRUCT
        PulseOnTime  : LREAL;
        PulseOffTime : LREAL;
    END_STRUCT
END_TYPE

// Machine/Components/Indicator/DUTs/HMI/ST_Indicator_HMI
TYPE
    ST_Indicator_HMI : STRUCT
        Config  : ST_Indicator_Config;
        Command : ST_Indicator_Command;
        Status  : ST_Indicator_Status;
    END_STRUCT
END_TYPE

// Machine/Components/Indicator/DUTs/HMI/ST_Indicator_Status
TYPE
    ST_Indicator_Status : STRUCT
        On       : BOOL;
        Off      : BOOL;
        Flashing : BOOL;
    END_STRUCT
END_TYPE

// Machine/Components/IRC5/DUTs/HMI/ST_IRC5_Command
TYPE
    ST_IRC5_Command : STRUCT
        Extend  : BOOL;
        Retract : BOOL;
    END_STRUCT
END_TYPE

// Machine/Components/IRC5/DUTs/HMI/ST_IRC5_Config
TYPE
    ST_IRC5_Config : STRUCT
        ExtendTime  : LREAL;
        RetractTime : LREAL;
    END_STRUCT
END_TYPE

// Machine/Components/IRC5/DUTs/HMI/ST_IRC5_HMI
TYPE
    ST_IRC5_HMI : STRUCT
        Config  : ST_MyComponent_Config;
        Command : ST_MyComponent_Command;
        Status  : ST_MyComponent_Status;
    END_STRUCT
END_TYPE

// Machine/Components/IRC5/DUTs/HMI/ST_IRC5_Status
TYPE
    ST_IRC5_Status : STRUCT
        Extended   : BOOL;
        Retracted  : BOOL;
        Extending  : BOOL;
        Retracting : BOOL;
    END_STRUCT
END_TYPE

// Machine/Components/IRC5/DUTs/ST_IRC5_Input
TYPE
    ST_IRC5_Input : STRUCT
        AutoMode          : BOOL;
        E_Stop            : BOOL;
        MotionSupervision : BOOL;
        MotorsOn          : BOOL;
        SignalsSimulated  : BOOL;
        AllTasksRunning   : BOOL;
        RunChainOK        : BOOL;
        PP_Moved          : BOOL;
    END_STRUCT
END_TYPE

// Machine/Components/IRC5/DUTs/ST_IRC5_IO
TYPE
    ST_IRC5_IO : STRUCT
        IN  : ST_IRC5_Input;
        OUT : ST_IRC5_Output;
    END_STRUCT
END_TYPE

// Machine/Components/IRC5/DUTs/ST_IRC5_Output
TYPE
    ST_IRC5_Output : STRUCT
        Pause      : BOOL;
        Resume     : BOOL;
        EStopReset : BOOL;
        MotorsOn   : BOOL;
        MotorsOff  : BOOL;
        PPtoMain   : BOOL;
    END_STRUCT
END_TYPE

// Machine/Components/Preplate_Rack/DUTs/E_RackState
{attribute 'qualified_only'}
{attribute 'strict'}
{attribute 'to_string'}
TYPE
    E_RackState : (
        Idle           := 0,
        CheckForBlock  := 10,
        CheckForLinked := 11,
        UnlockDoor     := 30,
        WaitForOpen    := 40,
        WaitForClose   := 50,
        LockDoor       := 60,
        DoorLockError  := 70,
        EnableDoor     := 80
    );
END_TYPE

// Machine/Components/Preplate_Rack/DUTs/linked_racks_typ
TYPE
    linked_racks_typ : STRUCT
        first_linked_rack  : INT;
        second_linked_rack : INT;
    END_STRUCT
END_TYPE

// Machine/Components/Preplate_Rack/DUTs/RackStateMachine
TYPE
    RackStateMachine : STRUCT
        nState       : INT;
        button_input : BOOL;
        button_light : BOOL;
        door_lock    : BOOL;
        door_closed  : BOOL;
        RisingEdge   : R_TRIG;
    END_STRUCT
END_TYPE

// Machine/Components/Preplate_Rack/DUTs/RackStatus
TYPE
    RackStatus : STRUCT
        available : BOOL;
        blocked   : BOOL;
    END_STRUCT
END_TYPE

// Machine/Components/Robot/DUTs/ST_Robot_Handshake_Input
TYPE
    ST_Robot_Handshake_Input : STRUCT
        SubStep           : BOOL;
        ErrorPresent      : BOOL;
        ServiceNumber     : USINT;
        MessageNumber     : UINT;
        Executing_Service : BOOL;
        Executing_Step    : BOOL;
        SubStepNumber     : E_WaitSync;
        ServiceComplete   : BOOL;
        StepComplete      : BOOL;
        TaskRunning       : BOOL;
    END_STRUCT
END_TYPE

// Machine/Components/Robot/DUTs/ST_Robot_Handshake_IO
TYPE
    ST_Robot_Handshake_IO : STRUCT
        IN  : ST_Robot_Handshake_Input;
        OUT : ST_Robot_Handshake_Output;
    END_STRUCT
END_TYPE

// Machine/Components/Robot/DUTs/ST_Robot_Handshake_Output
TYPE
    ST_Robot_Handshake_Output : STRUCT
        Abort              : BOOL;
        MessageSolution    : USINT;
        MessageAcknowledge : BOOL;
        SubStepResponse    : E_WaitSync;
        Execute_Service    : BOOL;
        Execute_Step       : BOOL;
        Execute_ServiceNum : USINT;
        Execute_StepNum    : UINT;
    END_STRUCT
END_TYPE

// Machine/Components/Template_MyComponent/DUTs/HMI/ST_MyComponent_Command
TYPE
    ST_MyComponent_Command : STRUCT
        Extend  : BOOL;
        Retract : BOOL;
    END_STRUCT
END_TYPE

// Machine/Components/Template_MyComponent/DUTs/HMI/ST_MyComponent_Config
TYPE
    ST_MyComponent_Config : STRUCT
        ExtendTime  : LREAL;
        RetractTime : LREAL;
    END_STRUCT
END_TYPE

// Machine/Components/Template_MyComponent/DUTs/HMI/ST_MyComponent_HMI
TYPE
    ST_MyComponent_HMI : STRUCT
        Config  : ST_MyComponent_Config;
        Command : ST_MyComponent_Command;
        Status  : ST_MyComponent_Status;
    END_STRUCT
END_TYPE

// Machine/Components/Template_MyComponent/DUTs/HMI/ST_MyComponent_Status
TYPE
    ST_MyComponent_Status : STRUCT
        Extended   : BOOL;
        Retracted  : BOOL;
        Extending  : BOOL;
        Retracting : BOOL;
    END_STRUCT
END_TYPE

// Machine/EquipmentModules/SamComm/DUTs/E_ContentType
{attribute 'qualified_only'}
{attribute 'strict'}
{attribute 'to_string'}
TYPE
    E_ContentType : (
        CT_NONE,
        CT_JSON,
        CT_CSV,
        CT_NOTASK,
        CT_NAK,
        CT_ACK,
        CT_MAX
    );
END_TYPE

// Machine/EquipmentModules/SamComm/DUTs/E_MessageCategory
{attribute 'qualified_only'}
{attribute 'strict'}
{attribute 'to_string'}
TYPE
    E_MessageCategory : (
        MC_NONE,
        MC_RFI,
        MC_INFO,
        MC_RFT,
        MC_TASK,
        MC_NOTASK,
        MC_STATUS,
        MC_STATUS_ACK,
        MC_NAK,
        MC_MAX
    );
END_TYPE

// Machine/EquipmentModules/SamComm/DUTs/E_MessageStatus
{attribute 'qualified_only'}
{attribute 'strict'}
{attribute 'to_string'}
TYPE
    E_MessageStatus : (
        MS_INIT,
        MS_BUSY,
        MS_RECEIVED,
        MS_SENT,
        MS_TIMED_OUT,
        MS_GOT_ACK,
        MS_GOT_NAK,
        MS_NO_DATA,
        MS_ERROR
    );
END_TYPE

// Machine/EquipmentModules/SamComm/DUTs/E_SAMCommStateMachine
{attribute 'qualified_only'}
{attribute 'strict'}
{attribute 'to_string'}
TYPE
    E_SAMCommStateMachine : (
        CREATE_RFI    := 0,
        SEND_RFI      := 1,
        WATCH_EVENTS  := 2,
        CREATE_STATUS := 3,
        SEND_STATUS   := 4,
        CREATE_RFT    := 5,
        SEND_RFT      := 6,
        PROCESS_REPLY := 7,
        CREATE_TASK   := 8,
        DISCONNECT    := 9,
        DISCONNECTING := 10,
        DEBUG         := 99

    );
END_TYPE

// Machine/EquipmentModules/SamComm/DUTs/E_TaskState
{attribute 'qualified_only'}
{attribute 'strict'}
{attribute 'to_string'}
TYPE
    E_TaskState : (
        IDLE,
        PENDING,
        ACTIVE,
        MANUAL,
        COMPLETE,
        ERROR,
        RECOVERY,
        ABORT,
        ABORT_RETRY,
        INVALID
    );
END_TYPE

// Machine/EquipmentModules/SamComm/DUTs/ST_Alert
TYPE
    ST_Alert : STRUCT
        Level   : STRING[10]; // Adjust size based on expected values (e.g., "WARNING")
        Message : STRING[50]; // Adjust size based on expected message lengths
    END_STRUCT
END_TYPE

// Machine/EquipmentModules/SamComm/DUTs/ST_Message
TYPE
    ST_Message : STRUCT
        content_type : E_ContentType;
        data         : STRING[1000];
        data_len     : UDINT;
        status       : E_MessageStatus;
    END_STRUCT
END_TYPE

// Machine/EquipmentModules/SamComm/DUTs/ST_Messages
TYPE
    ST_Messages : STRUCT
        MessageUuid     : STRING[40]; // UUIDs are typically 36 characters
        MessageCategory : STRING[20]; // E.g., "Status"
        TimeStamp       : STRING[12]; // Unsigned 64-bit integer for timestamp
        Status          : ST_Status;
    END_STRUCT
END_TYPE

// Machine/EquipmentModules/SamComm/DUTs/ST_PLC
TYPE
    ST_PLC : STRUCT
        State   : STRING[20]; // E.g., "SUSPENDED"
        Message : STRING[100]; // Adjust size based on expected message lengths
    END_STRUCT
END_TYPE

// Machine/EquipmentModules/SamComm/DUTs/ST_RFT
TYPE
    ST_RFT : STRUCT
        MessageUuid      : STRING[40]; // UUID string
        MessageCategory  : STRING[30]; // Adjust size as needed
        InResponseToUuid : STRING[40]; // Needs special handling to serialize as null
        TimeStamp        : STRING[12]; // Unsigned 64-bit integer for timestamp
        LineNumber       : INT; // Assuming line numbers are small integers
        StationName      : STRING[50]; // Adjust size as needed
        SubStation       : STRING[50]; // Adjust size as needed
        SubAsyncGroup    : STRING[50]; // Adjust size as needed
    END_STRUCT
END_TYPE

// Machine/EquipmentModules/SamComm/DUTs/ST_Status
TYPE
    ST_Status : STRUCT
        //Plc    : ST_Plc;//Sam doesn't do anything with this at the moment but can in the future
        Tasks : ARRAY[1..MAX_TASKS] OF ST_TaskStatus; // Array of 10 tasks
    //Alerts : ARRAY[1..2] OF ST_Alert; // Array of alerts but removing for now because sam doesn't do anything with the infomation provided ATM
    END_STRUCT
END_TYPE

// Machine/EquipmentModules/SamComm/DUTs/ST_Task
{attribute 'to_string'}
TYPE
    ST_Task : STRUCT
        Info          : ST_Task_Info;
        Data          : STRING[25000]; //Build Data from CSV/Json body from SAM
        CSV           : ST_CSV;
        StatusUpdate  : BOOL; // Send Status Update
        RFT_Requested : BOOL; // RFT Sent Out
        StepTimer     : TON; // Timer for 1-second delay    
    END_STRUCT
END_TYPE

// Machine/EquipmentModules/SamComm/DUTs/ST_Task_Info
{attribute 'to_string'}
TYPE
    ST_Task_Info : STRUCT
        State           : E_TaskState := E_TaskState.INVALID; // E.g., "active"
        TrussID         : STRING[50]; // Component ID
        CurrentTaskId   : UDINT; // 32-bit integer for task ID UDINT 0-4294967295
        LineNumber      : INT; // Assuming line numbers are small integers
        StationName     : STRING[50]; // Adjust size as needed
        SubStation      : STRING[50]; // Adjust size as needed
        TotalTaskSteps  : DINT; // Total number of steps in the task
        CurrentTaskStep : DINT; // Current step number
        Active          : BOOL;
    END_STRUCT
END_TYPE

// Machine/EquipmentModules/SamComm/DUTs/ST_TaskREF
TYPE
    ST_TaskREF : STRUCT
        Task : REFERENCE TO ST_Task;
    END_STRUCT
END_TYPE

// Machine/EquipmentModules/SamComm/DUTs/ST_TaskStatus
TYPE
    ST_TaskStatus : STRUCT
        State           : STRING; // E.g., "active"
        CurrentTaskId   : UDINT; // 32-bit integer for task ID UDINT 0-4294967295
        LineNumber      : INT; // Assuming line numbers are small integers
        StationName     : STRING[50]; // Adjust size as needed
        SubStation      : STRING[50]; // Adjust size as needed
        TotalTaskSteps  : DINT; // Total number of steps in the task
        CurrentTaskStep : DINT; // Current step number
    END_STRUCT
END_TYPE

// Machine/FunctionBlocks/Occupy Press Street/E_GateKeeperState
{attribute 'qualified_only'}
{attribute 'strict'}
{attribute 'to_string'}
TYPE
    E_GateKeeperState : (
        INVALID        := 0,
        IDLE           := 1,
        OCCUPIED_CAR_1 := 2,
        OCCUPIED_CAR_2 := 3,
        OCCUPIED_CAR_3 := 4,
        OCCUPIED_ROBOT := 5,
        RESET          := 6,
        ERROR          := 7
    );
END_TYPE

// Machine/FunctionBlocks/Occupy Press Street/ST_MediatorInterface
TYPE
    ST_MediatorInterface : STRUCT
        Request    : BOOL;
        Permission : BOOL;
    END_STRUCT
END_TYPE

// GVLs/Global
VAR_GLOBAL
    // change speeds of motors 

    AutoMode : BOOL := TRUE;

    // Bell Evermen point backup

    BEPoint_Backup : ST_BEPointDefinitions;

    // Sys Config backup values

    Sys_Config : ST_SysConfig;

    //trigger all message boxes

    testmessagebox : BOOL;

    DOUBLEPICK_MIN_LENGTH : LREAL;
	
	BoardToleranceRatio_short : LREAL := 0.0155;

    BoardToleranceRatio_med : LREAL := 0.021;

    BoardToleranceRatio_long : LREAL := 0.0249;

    BoardAcceptanceTolerance_mm : LREAL := 25;

// 
//     BoardToleranceRatio_short : LREAL := 0.0039;
// 
//     BoardToleranceRatio_med : LREAL := 0.0132;
// 
//     BoardToleranceRatio_long : LREAL := 0.0135;
// 
//     BoardAcceptanceTolerance_mm : LREAL := 10;

END_VAR

VAR_GLOBAL CONSTANT
    // Max number of commands we are able to receive in a JSON file

    MAX_COMMAND_COUNT : UDINT := 12;

    // Max number of steps we can see in a JSON file

    MAX_STEP_COUNT   : UDINT := 300;
    MAX_DETAIL_COUNT : UDINT := 35;
    MAX_DATA_COUNT   : UDINT := 20;

    // Max number of details we can receive in a JSON file

    MAX_POSITIONS : UDINT := 10;

    //Max number of material we expect to see per conveyor

    MAX_OUTFEED_MATERIAL : UDINT := 50;

    MAX_NUMBER_OF_BOARDS : UDINT := MAX_STEP_COUNT;

    MAX_NUMBER_OF_PLATES : UDINT := 50;

    MAX_NUMBER_OF_POSITIONS : UDINT := MAX_POSITIONS;

    //max number of alarms by default on EquipmentModule_SR and CustomComponents

    MAX_ALARM_COUNT : UDINT := 6;

    BOARD_LENGTH_SENSOR1_LOCATION : LREAL := 2652.7125;

    BOARD_LENGTH_SENSOR2_LOCATION : LREAL := 5092.7;

    MAX_BOARDLEN_LIM : LREAL := 3200;

    MAX_TASKS : INT := 4;

    PLCPRJ_BUFFER_SIZE : UDINT := 262144; (* Max. internal fifo/receiver buffer size *)

    PLCPRJ_CLIENT_SEND_CYCLE_TIME : TIME := T#5S;
    PLCPRJ_RECEIVE_POLLING_TIME   : TIME := T#100MS;
    PLCPRJ_RECEIVE_TIMEOUT        : TIME := T#30S;

    (* Some project specific error codes *)

    PLCPRJ_ERROR_RECEIVE_TIMEOUT   : UDINT := 16#8101; (* Receive timeout *)
    PLCPRJ_ERROR_SENDFIFO_OVERFLOW : UDINT := 16#8102; (* Send fifo overflow *)
    PLCPRJ_ERROR_RECFIFO_OVERFLOW  : UDINT := 16#8103; (* Receive fifo overflow *)

    PICK_DEVICE_WIDTH   : REAL := 203;
    DEFAULT_PICK_OFFSET : REAL := 200;

END_VAR

// Version/Global_Version
{attribute 'TcGenerated'}
{attribute 'no-analysis'}
{attribute 'linkalways'}
// This function has been automatically generated from the project information.
VAR_GLOBAL CONSTANT
	{attribute 'const_non_replaced'}
	stLibVersion_RoofTrussLibrary : ST_LibVersion := (iMajor := 0, iMinor := 1, iBuild := 0, iRevision := 0, nFlags := 0, sVersion := '0.1.0.0');
END_VAR

// Machine/Components/BasicSlaveAxis_SOE/FB_Component_BasicSlaveAxis_SoE
FUNCTION_BLOCK FB_Component_BasicSlaveAxis_SoE EXTENDS FB_Component_BasicSlaveAxis IMPLEMENTS I_BasicAxis
VAR
    DriveReset  : FB_ResetRoutine_SoEDrive;
    State_Reset : INT;
    HomingInfo  : ST_HomingParams;

END_VAR

METHOD CyclicLogic
DriveReset.Axis := THIS^;
DriveReset.CyclicLogic();

SUPER^.CyclicLogic();
END_METHOD

(*! @summary Clears error flags and error IDs for this component*)
METHOD Reset : BOOL
Reset := FALSE;

IF _Error THEN
    CASE State_Reset OF
        0:
            DriveReset.Execute();
            State_Reset := State_Reset + 10;
            Trace('Drive Reset Called ');

        10:
            IF NOT DriveReset.Busy THEN
                State_Reset := State_Reset + 10;
                Trace('Drive Reset Done ');
            END_IF

        20:
            IF SUPER^.Reset() THEN
                Reset       := TRUE;
                State_Reset := 0;
            END_IF
    END_CASE
ELSE
    IF SUPER^.Reset() THEN
        Reset := TRUE;
    END_IF
END_IF
END_METHOD

END_FUNCTION_BLOCK

// Machine/Components/Button/FB_Component_Button
FUNCTION_BLOCK FB_Component_Button EXTENDS FB_ComponentBase_SR
VAR
    Button : FB_DigitalSensor := (Name := 'Button');
    LED    : FB_Component_Indicator;

END_VAR

//! @summary This method serves as the entry point for all underlying FB logic
METHOD PUBLIC CyclicLogic

//! @description This method should be called cyclically by descendant function blocks by invoking <c>SUPER^.CyclicLogic()</c>.  Alternatively, the contents of this method could be reimplemented entirely in which case a call to this method would not be necessary.
// Initialise Component

IF NOT _InitComplete THEN
    _InitComplete := Initialize();
    RETURN;
END_IF

//Custom Component Logic goes here

// Call Super

SUPER^.CyclicLogic();

// Set Current Alarm Severity

_CurrentAlarmSeverity := F_GetMaxSeverityRaised(Alarms := Comp_Alarms, CurrentSeverity := _CurrentAlarmSeverity);

Button.CyclicLogic();
LED.CyclicLogic();
END_METHOD

METHOD PROTECTED CreateEvents
VAR_INPUT
END_VAR
SUPER^.CreateEvents();
END_METHOD

//! @summary Basic component initialization logic
METHOD PROTECTED Initialize : BOOL;

//! @description This method is called by <c>CyclicLogic()</c> as required
CreateEvents();

IF SUPER^.Initialize() THEN
    Initialize := TRUE;
END_IF
END_METHOD

METHOD PROTECTED Monitoring
VAR_INPUT
END_VAR
SUPER^.Monitoring();
END_METHOD

PROPERTY Button_Pressed : bool
GET
Button_Pressed := Button.Active;
END_GET
END_PROPERTY

END_FUNCTION_BLOCK

// Machine/Components/ComponentBase_SR/FB_ComponentBase_SR
FUNCTION_BLOCK FB_ComponentBase_SR EXTENDS FB_ComponentBase
VAR_INPUT
END_VAR

VAR_OUTPUT
END_VAR

VAR
    Comp_Alarms : ARRAY[1..20] OF FB_TcAlarm;

    i : UDINT;

END_VAR

METHOD ClearAlarms
VAR_INPUT
    MyAlarms : ARRAY[1..Global.MAX_ALARM_COUNT] OF FB_TcAlarm;
END_VAR

VAR
    i : UDINT;
END_VAR
FOR i := 1 TO Global.MAX_ALARM_COUNT DO
    MyAlarms[i].Clear(0, 0);
END_FOR;
END_METHOD

METHOD RaiseAlarm2Args
VAR_IN_OUT
    fbAlarm : FB_TcAlarm; //Alarm to be raised
END_VAR

VAR_INPUT
    String_1 : STRING; //First String Parameter (The Name of this component will be applied first automatically)
    String_2 : STRING; //Second String Parameter
END_VAR
F_RaiseAlarmWithStringParameters(Alarm := fbAlarm, String_1 := Name, String_2 := String_1, String_3 := String_2);
END_METHOD

METHOD Reset : BOOL
_Error   := FALSE;
_ErrorID := 0;

IF SUPER^.Reset() THEN
    Reset := TRUE;
END_IF
END_METHOD

END_FUNCTION_BLOCK

// Machine/Components/Indicator/FB_Component_Indicator
FUNCTION_BLOCK FB_Component_Indicator EXTENDS FB_ComponentBase_SR IMPLEMENTS I_Indicator
VAR

    // Outputs

    IndicatorOutput AT %Q* : BOOL;

    // HMI

    Indicator_HMI : ST_Indicator_HMI;

    // Alarms

    IndicatorAlarms : ARRAY[1..Indicator_ALARMS_COUNT] OF FB_TcAlarm;

    // Internal variables

    Pulse     : FB_PulseGenerator;
    _Flashing : BOOL;
    _On       : BOOL;

END_VAR

VAR CONSTANT
    Indicator_ALARMS_COUNT : UDINT := 5;
END_VAR

//! @summary This method serves as the entry point for all underlying FB logic
METHOD PUBLIC CyclicLogic

//! @description This method should be called cyclically by descendant function blocks by invoking <c>SUPER^.CyclicLogic()</c>.  Alternatively, the contents of this method could be reimplemented entirely in which case a call to this method would not be necessary.
// Initialise Component

IF NOT _InitComplete THEN
    _InitComplete := Initialize();
    RETURN;
END_IF

IF _Flashing THEN
    Pulse.CyclicLogic();
    IndicatorOutput := Pulse.PulseOutput;
END_IF

// Call Super

SUPER^.CyclicLogic();

// Set Current Alarm Severity

_CurrentAlarmSeverity := F_GetMaxSeverityRaised(Alarms := IndicatorAlarms, CurrentSeverity := _CurrentAlarmSeverity);
END_METHOD

METHOD PROTECTED CreateEvents
VAR_INPUT
END_VAR
F_CreateAllEventsInClass(Alarms     := IndicatorAlarms,
                         ClassSize  := SIZEOF(TC_EVENTS.ComponentBase),
                         pInitEvent := ADR(TC_EVENTS.ComponentBase.InitReferenceEvent),
                         Prefix     := _Name);

SUPER^.CreateEvents();
END_METHOD

METHOD Flash
_Flashing := TRUE;
_On       := FALSE;

IndicatorOutput := Pulse.PulseOutput;
END_METHOD

//! @summary Basic component initialization logic
METHOD PROTECTED Initialize : BOOL;

//! @description This method is called by <c>CyclicLogic()</c> as required
CreateEvents();

IF SUPER^.Initialize() THEN
    Initialize := TRUE;
END_IF
END_METHOD

METHOD PROTECTED Monitoring
VAR_INPUT
END_VAR
IF NOT IndicatorAlarms[E_ComponentBase.SimulationWarning].bRaised AND _Simulate AND NOT Parameters_BaseComponent.INHIBIT_SIMULATION_WARNING THEN
    IndicatorAlarms[E_ComponentBase.SimulationWarning].Raise(0);
ELSIF IndicatorAlarms[E_ComponentBase.SimulationWarning].bRaised AND NOT _Simulate THEN
    IndicatorAlarms[E_ComponentBase.SimulationWarning].Clear(0, 0);
END_IF

_CurrentAlarmSeverity := TcEventSeverity.Verbose;
_CurrentAlarmSeverity := F_GetMaxSeverityRaised(Alarms := IndicatorAlarms, CurrentSeverity := _CurrentAlarmSeverity);

SUPER^.Monitoring();
END_METHOD

METHOD Reset : BOOL
TurnOff();
END_METHOD

METHOD TurnOff
_Flashing := FALSE;
_On       := FALSE;

IndicatorOutput := FALSE;
END_METHOD

METHOD TurnOn
_Flashing := FALSE;
_On       := TRUE;

IndicatorOutput := TRUE;
END_METHOD

PROPERTY Flashing : BOOL
GET
Flashing := _Flashing;
END_GET
END_PROPERTY

PROPERTY Off : BOOL
GET
Off := NOT _ON AND NOT _Flashing;
END_GET
END_PROPERTY

PROPERTY PUBLIC OffTime : TIME
SET
Pulse.OffTime := OffTime;
END_SET
END_PROPERTY

PROPERTY On : BOOL
GET
On := _On;
END_GET
END_PROPERTY

PROPERTY PUBLIC OnTime : TIME
SET
Pulse.OnTime := OnTime;
END_SET
END_PROPERTY

END_FUNCTION_BLOCK

// Machine/Components/Indicator/Interfaces/I_Indicator
INTERFACE I_Indicator

METHOD Flash
VAR_INPUT
END_VAR
END_METHOD

METHOD TurnOff
VAR_INPUT
END_VAR
END_METHOD

METHOD TurnOn
VAR_INPUT
END_VAR
END_METHOD

END_INTERFACE

// Machine/FunctionBlocks/PulseGenerator/FB_PulseGenerator
FUNCTION_BLOCK FB_PulseGenerator
VAR
    PulseOn_TON  : TON;
    PulseOff_TON : TON;
    R_TRIG_0     : R_TRIG;
    Pulse_TON    : TON;
    OutRS        : RS;
    _OnTime      : TIME := T#500MS;
    _OffTime     : TIME := T#500MS;
    _PulseOutput : BOOL;
END_VAR

METHOD CyclicLogic
PulseOn_TON(IN := PulseOutput, PT := _OnTime);
PulseOff_TON(IN := NOT (PulseOutput), PT := _OffTime);
OutRS(SET := PulseOff_TON.Q, RESET1 := PulseOn_TON.Q);
_PulseOutput := OutRS.Q1;
END_METHOD

PROPERTY OffTime : TIME
SET
_OffTime := OffTime;
END_SET
END_PROPERTY

PROPERTY OnTime : TIME
SET
_OnTime := OnTime;
END_SET
END_PROPERTY

PROPERTY PulseOutput : BOOL
GET
PulseOutput := _PulseOutput;
END_GET
END_PROPERTY

END_FUNCTION_BLOCK

// Machine/Components/ComponentBase_SR/Interfaces/I_ComponentBase_SR
INTERFACE I_ComponentBase_SR

END_INTERFACE

// Machine/Components/ControlPendant/FB_ControlPendant
FUNCTION_BLOCK FB_ControlPendant EXTENDS FB_ComponentBase_SR
VAR
    KeySwitch_Idle    : FB_DigitalSensor := (Name := 'KeySwitch_Idle'); // Auto mode key switch
    KeySwitch_Auto    : FB_DigitalSensor := (Name := 'KeySwitch_Auto'); // Manual mode forward
    KeySwitch_Manual1 : FB_DigitalSensor := (Name := 'KeySwitch_Manual1'); // Manual mode reverse
    KeySwitch_Manual2 : FB_DigitalSensor := (Name := 'KeySwitch_Manual2'); // Manual mode reverse

    GreenButton  : FB_Component_Button := (Name := 'GreenButton');
    YellowButton : FB_Component_Button := (Name := 'YellowButton');
    BlueButton   : FB_Component_Button := (Name := 'BlueButton');

END_VAR

//! @summary This method serves as the entry point for all underlying FB logic
METHOD PUBLIC CyclicLogic

//! @description This method should be called cyclically by descendant function blocks by invoking <c>SUPER^.CyclicLogic()</c>.  Alternatively, the contents of this method could be reimplemented entirely in which case a call to this method would not be necessary.
// Initialise Component

IF NOT _InitComplete THEN
    _InitComplete := Initialize();
    RETURN;
END_IF

//Custom Component Logic goes here

// Call Super

SUPER^.CyclicLogic();

// Set Current Alarm Severity

_CurrentAlarmSeverity := F_GetMaxSeverityRaised(Alarms := Comp_Alarms, CurrentSeverity := _CurrentAlarmSeverity);

KeySwitch_Idle.CyclicLogic();
KeySwitch_Auto.CyclicLogic();
KeySwitch_Manual1.CyclicLogic();
KeySwitch_Manual2.CyclicLogic();

GreenButton.CyclicLogic();
YellowButton.CyclicLogic();
BlueButton.CyclicLogic();
END_METHOD

METHOD PROTECTED CreateEvents
VAR_INPUT
END_VAR
SUPER^.CreateEvents();
END_METHOD

//! @summary Basic component initialization logic
METHOD PROTECTED Initialize : BOOL;

//! @description This method is called by <c>CyclicLogic()</c> as required
CreateEvents();

IF SUPER^.Initialize() THEN
    Initialize := TRUE;
END_IF
END_METHOD

METHOD PROTECTED Monitoring
VAR_INPUT
END_VAR
SUPER^.Monitoring();
END_METHOD

PROPERTY Mode_Auto : bool
GET
Mode_Auto := KeySwitch_Auto.Active;
END_GET
END_PROPERTY

PROPERTY Mode_Idle : bool
GET
Mode_Idle := NOT (KeySwitch_Auto.Active AND KeySwitch_Manual1.Active AND KeySwitch_Manual2.Active);
END_GET
END_PROPERTY

PROPERTY Mode_Manual_1 : bool
GET
Mode_Manual_1 := KeySwitch_Manual1.Active;
END_GET
END_PROPERTY

PROPERTY Mode_Manual_2 : bool
GET
Mode_Manual_2 := KeySwitch_Manual2.Active;
END_GET
END_PROPERTY

END_FUNCTION_BLOCK

// Machine/Components/ControlPendant/FB_ControlPendant_Outfeed
FUNCTION_BLOCK FB_ControlPendant_Outfeed EXTENDS FB_ComponentBase_SR
VAR
    Light           : FB_Component_Indicator := (Name := 'Pendant Light');
    SafetyReset     : FB_Component_Button    := (Name := 'Oufeed Safety Reset');
    ClearConveyor   : FB_Component_Button    := (Name := 'Clear Conveyor');
    RetractSlideout : FB_Component_Button    := (Name := 'Retract Slideout');
    ExtendSlideout  : FB_Component_Button    := (Name := 'Extend Slideout');

END_VAR

//! @summary This method serves as the entry point for all underlying FB logic
METHOD PUBLIC CyclicLogic

//! @description This method should be called cyclically by descendant function blocks by invoking <c>SUPER^.CyclicLogic()</c>.  Alternatively, the contents of this method could be reimplemented entirely in which case a call to this method would not be necessary.
// Initialise Component

IF NOT _InitComplete THEN
    _InitComplete := Initialize();
    RETURN;
END_IF

//Custom Component Logic goes here

// Call Super

SUPER^.CyclicLogic();

// Set Current Alarm Severity

_CurrentAlarmSeverity := F_GetMaxSeverityRaised(Alarms := Comp_Alarms, CurrentSeverity := _CurrentAlarmSeverity);

Light.CyclicLogic();
SafetyReset.CyclicLogic();
ClearConveyor.CyclicLogic();
RetractSlideout.CyclicLogic();
ExtendSlideout.CyclicLogic();
END_METHOD

METHOD PROTECTED CreateEvents
VAR_INPUT
END_VAR
SUPER^.CreateEvents();
END_METHOD

//! @summary Basic component initialization logic
METHOD PROTECTED Initialize : BOOL;

//! @description This method is called by <c>CyclicLogic()</c> as required
CreateEvents();

IF SUPER^.Initialize() THEN
    Initialize := TRUE;
END_IF
END_METHOD

METHOD PROTECTED Monitoring
VAR_INPUT
END_VAR
SUPER^.Monitoring();
END_METHOD

END_FUNCTION_BLOCK

// Machine/Components/Conveyor/FB_Conveyor
FUNCTION_BLOCK FB_Conveyor EXTENDS FB_Component_BasicSlaveAxis_SoE

VAR CONSTANT
    CONVEYOR_ALARMS_COUNT : USINT := 10;
END_VAR

VAR
    ConveyorAlarms : ARRAY[1..CONVEYOR_ALARMS_COUNT] OF FB_TcAlarm;

END_VAR

METHOD CyclicLogic
SUPER^.CyclicLogic();
END_METHOD

METHOD AlarmRaiseBasic : BOOL
VAR_INPUT
    alarm : E_OutfeedConveyor;
    raise : BOOL;
END_VAR
IF (NOT ConveyorAlarms[alarm].bRaised) AND raise THEN
    // Raise alarm if we are NOT in auto
    ConveyorAlarms[alarm].Raise(0);
ELSIF ConveyorAlarms[alarm].bRaised AND NOT raise THEN
    // Clear alarm if we return to auto
    ConveyorAlarms[alarm].Clear(0, 0);
END_IF;
END_METHOD

METHOD PROTECTED CreateEvents
VAR_INPUT
END_VAR
// F_CreateAllEventsInClass(Alarms		:= ConveyorAlarms,
// 						 ClassSize	:= SIZEOF(TC_EVENTS.OutfeedConveyor),
// 						 pInitEvent := ADR(TC_EVENTS.OutfeedConveyor.InitReferenceEvent),
// 						 Prefix		:= _Name);
SUPER^.CreateEvents();
END_METHOD

METHOD PROTECTED Monitoring
VAR_INPUT
END_VAR
// AlarmRaiseBasic(alarmlist := ConveyorAlarms,alarm := E_OutfeedConveyor.NoTrussData,NoTrussDataAlarm);

//////////////////////////////////////////////////////////////////////////
// Wrap-up: Evaluate overall severity, then run the extended Monitoring
//////////////////////////////////////////////////////////////////////////
_CurrentAlarmSeverity := TcEventSeverity.Verbose;
_CurrentAlarmSeverity := F_GetMaxSeverityRaised(Alarms := ConveyorAlarms, CurrentSeverity := _CurrentAlarmSeverity);

// Finally, run the extended monitoring
SUPER^.Monitoring();
END_METHOD

METHOD SimHoming : BOOL
VAR_INPUT
    Motor  : REFERENCE TO FB_Component_BasicSlaveAxis_SoE;
    SimPos : LREAL;
END_VAR

VAR_INST
    _SimHomingState : USINT;
    _SetPositionSim : FB_HomeRoutine_SetPosition;
    Timeout_TON     : TON;
    TimeoutCount    : USINT;
END_VAR
CASE _SimHomingState OF
    0:
        SimHoming                    := FALSE;
        Motor.HomeMethod             := _SetPositionSim;
        _SetPositionSim.HomePosition := SimPos;
        _SetPositionSim.Execute();
        _SimHomingState := 10;
        Timeout_TON(IN := FALSE, PT := T#500MS);

    10:
        Timeout_TON(IN := TRUE, PT := T#500MS);

        IF _SetPositionSim.Busy = FALSE AND ABS(Motor.ActualPosition - SimPos) < 1 THEN
            _SimHomingState := 20;
        END_IF

        IF Timeout_TON.Q THEN

            IF TimeoutCount <= 3 THEN
                _SimHomingState := 0;
                TimeoutCount    := TimeoutCount + 1;
            ELSE
                _SimHomingState := 15;
            END_IF
        END_IF

    15:

        //Warning, Home didn't work
    20:
        SimHoming       := TRUE;
        _SimHomingState := 0;
        TimeoutCount    := 0;
END_CASE
END_METHOD

PROPERTY ParentResponseDefinitions : ARRAY[0..4] OF E_AlarmResponse
GET
ParentResponseDefinitions[TcEventSeverity.Verbose]  := E_AlarmResponse.NoResponse;
ParentResponseDefinitions[TcEventSeverity.Info]     := E_AlarmResponse.NoResponse;
ParentResponseDefinitions[TcEventSeverity.Warning]  := E_AlarmResponse.NoResponse;
ParentResponseDefinitions[TcEventSeverity.Error]    := E_AlarmResponse.NoResponse;
ParentResponseDefinitions[TcEventSeverity.Critical] := E_AlarmResponse.Suspend_Immediate;
END_GET
END_PROPERTY

END_FUNCTION_BLOCK

// Machine/Components/DoubleSolenoidRetractFeedback/FB_DoubleSolenoidRetractFeedback
FUNCTION_BLOCK FB_DoubleSolenoidRetractFeedback EXTENDS FB_DoubleSolenoid
VAR
    RetractedSensor AT %I* : BOOL;
END_VAR

METHOD PROTECTED Feedback
IF NOT _Simulate THEN
    _Extended  := NOT RetractedSensor;
    _Retracted := RetractedSensor;
    Extend_TON(IN := _Extending, PT := LREAL_TO_TIME(_ExtendTime));
    Retract_TON(IN := _Retracting, PT := LREAL_TO_TIME(_RetractTime));

    IF Extend_TON.Q AND RetractedSensor THEN
        IF NOT SolenoidAlarms[E_CylinderAlarms.ExtendTimeout].bRaised THEN
            SolenoidAlarms[E_CylinderAlarms.ExtendTimeout].Raise(0);
            _ExtendRequest := FALSE;
            _Extending     := FALSE;
        END_IF
    ELSIF _Extending AND NOT RetractedSensor THEN
        _Extended  := TRUE;
        _Extending := FALSE;
    END_IF

    IF Retract_TON.Q AND NOT RetractedSensor THEN
        IF NOT SolenoidAlarms[E_CylinderAlarms.RetractTimeout].bRaised THEN
            SolenoidAlarms[E_CylinderAlarms.RetractTimeout].Raise(0);
            _RetractRequest := FALSE;
            _Retracting     := FALSE;
        END_IF
    ELSIF _Retracting AND RetractedSensor THEN
        _Retracted  := TRUE;
        _Retracting := FALSE;
    END_IF
ELSE
    SUPER^.Feedback();
END_IF
END_METHOD

METHOD PROTECTED HardwareInit
IF NOT RetractedSensor THEN
    _Extended  := TRUE;
    _Retracted := FALSE;
ELSIF RetractedSensor THEN
    _Extended  := FALSE;
    _Retracted := TRUE;
END_IF
END_METHOD

PROPERTY RetractedInput : BOOL
SET
RetractedSensor := RetractedInput;
END_SET
END_PROPERTY

END_FUNCTION_BLOCK

// Machine/Components/DualChannelIndicator/FB_DualChannelMonitor
FUNCTION_BLOCK FB_DualChannelMonitor EXTENDS FB_ComponentBase_SR
VAR
    CH_1 : FB_DigitalSensor := (Name := 'Channel_1'); // Auto mode key switch
    CH_2 : FB_DigitalSensor := (Name := 'Channel_1'); // Manual mode forward
    LED  : FB_Component_Indicator := (Name := 'LED'); // LED if available
	SIM_ResetChannels: BOOL;
	
	Sim_Reset_R_TRIG : R_TRIG;
END_VAR

//! @summary This method serves as the entry point for all underlying FB logic
METHOD PUBLIC CyclicLogic

//! @description This method should be called cyclically by descendant function blocks by invoking <c>SUPER^.CyclicLogic()</c>.  Alternatively, the contents of this method could be reimplemented entirely in which case a call to this method would not be necessary.
// Initialise Component

IF NOT _InitComplete THEN
    _InitComplete := Initialize();
    RETURN;
END_IF

//Custom Component Logic goes here

// Call Super

SUPER^.CyclicLogic();

// Set Current Alarm Severity

_CurrentAlarmSeverity := F_GetMaxSeverityRaised(Alarms := Comp_Alarms, CurrentSeverity := _CurrentAlarmSeverity);

CH_1.CyclicLogic();
CH_2.CyclicLogic();

CH_1.InSimulation := _Simulate;
CH_2.InSimulation := _Simulate;

Sim_Reset_R_TRIG(CLK := _Simulate);
IF Sim_Reset_R_TRIG.Q THEN
	SIM_ResetChannels := TRUE;
END_IF

IF SIM_ResetChannels THEN
    CH_1.SimulationInput := TRUE;
    CH_2.SimulationInput := TRUE;
ELSE
    CH_1.SimulationInput := FALSE;
    CH_2.SimulationInput := FALSE;
END_IF

LED.CyclicLogic();
END_METHOD

METHOD PROTECTED CreateEvents
VAR_INPUT
END_VAR
SUPER^.CreateEvents();
END_METHOD

//! @summary Basic component initialization logic
METHOD PROTECTED Initialize : BOOL;

//! @description This method is called by <c>CyclicLogic()</c> as required
CreateEvents();

IF SUPER^.Initialize() THEN
    Initialize := TRUE;
END_IF
END_METHOD

PROPERTY BothChannelsOK : BOOL
GET
BothChannelsOK := CH_1.Active AND CH_2.Active;
END_GET
END_PROPERTY

END_FUNCTION_BLOCK

// Machine/Components/IRC5/Interfaces/I_IRC5
INTERFACE I_IRC5

END_INTERFACE

// Machine/Components/IRC5/FB_Component_IRC5
FUNCTION_BLOCK FB_Component_IRC5 EXTENDS FB_ComponentBase_SR IMPLEMENTS I_IRC5

VAR
    ControllerIO : ST_IRC5_IO;
    Pulse        : FB_PulseGenerator;
    // Inputs

    InputArray AT %I* : ARRAY[0..1] OF USINT;

    // Outputs

    OutputArray AT %Q* : ARRAY[0..1] OF USINT;

    // HMI

    IRC5_HMI : ST_IRC5_HMI;

    // Alarms

    IRC5Alarms : ARRAY[1..IRC5_ALARMS_COUNT] OF FB_TcAlarm;

    _Start_State : INT;
    _Reset_State : INT;
END_VAR

VAR CONSTANT
    IRC5_ALARMS_COUNT : UDINT := 14;
END_VAR

//! @summary This method serves as the entry point for all underlying FB logic
METHOD PUBLIC CyclicLogic

//! @description This method should be called cyclically by descendant function blocks by invoking <c>SUPER^.CyclicLogic()</c>.  Alternatively, the contents of this method could be reimplemented entirely in which case a call to this method would not be necessary.
// Initialise Component

IF NOT _InitComplete THEN
    _InitComplete := Initialize();
    RETURN;
END_IF

Pulse.CyclicLogic();

SignalMapping();
Monitoring(); //Constant error and status monitoring

// Call Super

SUPER^.CyclicLogic();

// Set Current Alarm Severity

_CurrentAlarmSeverity := F_GetMaxSeverityRaised(Alarms := Comp_Alarms, CurrentSeverity := _CurrentAlarmSeverity);
END_METHOD

METHOD Abort : BOOL
VAR_INPUT
END_VAR
Abort := FALSE;

IF _Simulate THEN
    Abort := TRUE;
    RETURN;
END_IF

IF Stop() THEN
    ControllerIO.OUT.PPtoMain := Pulse.PulseOutput;

    IF ControllerIO.IN.PP_Moved THEN
        ControllerIO.OUT.PPtoMain := FALSE;
        Abort                     := TRUE;
        Trace('IRC5 Abort Finished ');
    END_IF
END_IF
END_METHOD

METHOD PROTECTED CreateEvents
VAR_INPUT
END_VAR
F_CreateAllEventsInClass(Alarms     := IRC5Alarms,
                         ClassSize  := SIZEOF(TC_EVENTS.IRC5),
                         pInitEvent := ADR(TC_EVENTS.IRC5.InitReferenceEvent),
                         Prefix     := _Name);

SUPER^.CreateEvents();
END_METHOD

METHOD EStopReset : BOOL
VAR_INPUT
END_VAR
IF ControllerIO.IN.AllTasksRunning OR _Simulate THEN
    EStopReset := TRUE;
    RETURN;
END_IF

EStopReset := FALSE;

CASE _Reset_State OF
    0:

        IF NOT ControllerIO.IN.E_Stop THEN
            _Reset_State := 2;
        ELSIF ControllerIO.IN.RunChainOK THEN
            _Reset_State := 2;
        END_IF

    1:
        ControllerIO.OUT.EStopReset := Pulse.PulseOutput;

        IF ControllerIO.IN.E_Stop = TRUE THEN
            ControllerIO.OUT.EStopReset := FALSE;
            _Reset_State                := 2;
        END_IF

    2:
        EStopReset   := TRUE;
        _Reset_State := 0;
END_CASE
END_METHOD

//! @summary Basic component initialization logic
METHOD PROTECTED Initialize : BOOL;

//! @description This method is called by <c>CyclicLogic()</c> as required
CreateEvents();

IF SUPER^.Initialize() THEN
    Initialize := TRUE;
END_IF
END_METHOD

METHOD PROTECTED Monitoring
VAR_INPUT
END_VAR
///////////////////////////////////////////////////////////////////////////////
// 5. Auto: ID=5
///////////////////////////////////////////////////////////////////////////////
IF (NOT IRC5Alarms[E_IRC5.Auto].bRaised) AND (NOT ControllerIO.IN.AutoMode) THEN
    // Raise alarm if we are NOT in auto
    IRC5Alarms[E_IRC5.Auto].Raise(0);
ELSIF IRC5Alarms[E_IRC5.Auto].bRaised AND (ControllerIO.IN.AutoMode) THEN
    // Clear alarm if we return to auto
    IRC5Alarms[E_IRC5.Auto].Clear(0, 0);
END_IF;

///////////////////////////////////////////////////////////////////////////////
// 6. Estop: ID=6
///////////////////////////////////////////////////////////////////////////////
IF (NOT IRC5Alarms[E_IRC5.Estop].bRaised) AND (NOT ControllerIO.IN.E_Stop) THEN
    IRC5Alarms[E_IRC5.Estop].Raise(0);
ELSIF IRC5Alarms[E_IRC5.Estop].bRaised AND (ControllerIO.IN.E_Stop) THEN
    IRC5Alarms[E_IRC5.Estop].Clear(0, 0);
END_IF;

///////////////////////////////////////////////////////////////////////////////
// 7. MotorSupervision: ID=7
///////////////////////////////////////////////////////////////////////////////
IF (NOT IRC5Alarms[E_IRC5.MotorSupervision].bRaised) AND (NOT ControllerIO.IN.MotionSupervision) THEN
    IRC5Alarms[E_IRC5.MotorSupervision].Raise(0);
ELSIF IRC5Alarms[E_IRC5.MotorSupervision].bRaised AND (ControllerIO.IN.MotionSupervision) THEN
    IRC5Alarms[E_IRC5.MotorSupervision].Clear(0, 0);
END_IF;

///////////////////////////////////////////////////////////////////////////////
// 8. MotorsOn: ID=8
///////////////////////////////////////////////////////////////////////////////
IF (NOT IRC5Alarms[E_IRC5.MotorsOn].bRaised) AND (ControllerIO.IN.MotorsOn) THEN
    IRC5Alarms[E_IRC5.MotorsOn].Raise(0);
ELSIF IRC5Alarms[E_IRC5.MotorsOn].bRaised AND (NOT ControllerIO.IN.MotorsOn) THEN
    IRC5Alarms[E_IRC5.MotorsOn].Clear(0, 0);
END_IF;

///////////////////////////////////////////////////////////////////////////////
// 9. SignalsSimulated: ID=9
///////////////////////////////////////////////////////////////////////////////
IF (NOT IRC5Alarms[E_IRC5.SignalsSimulated].bRaised) AND (NOT ControllerIO.IN.SignalsSimulated) THEN
    IRC5Alarms[E_IRC5.SignalsSimulated].Raise(0);
ELSIF IRC5Alarms[E_IRC5.SignalsSimulated].bRaised AND (ControllerIO.IN.SignalsSimulated) THEN
    IRC5Alarms[E_IRC5.SignalsSimulated].Clear(0, 0);
END_IF;

///////////////////////////////////////////////////////////////////////////////
// 10. AllTasksRunning: ID=10
///////////////////////////////////////////////////////////////////////////////
IF (NOT IRC5Alarms[E_IRC5.AllTasksRunning].bRaised) AND (ControllerIO.IN.AllTasksRunning) THEN
    IRC5Alarms[E_IRC5.AllTasksRunning].Raise(0);
ELSIF IRC5Alarms[E_IRC5.AllTasksRunning].bRaised AND (NOT ControllerIO.IN.AllTasksRunning) THEN
    IRC5Alarms[E_IRC5.AllTasksRunning].Clear(0, 0);
END_IF;

///////////////////////////////////////////////////////////////////////////////
// 11. AllTasksNotRunning: ID=11
///////////////////////////////////////////////////////////////////////////////
// Raise if tasks are NOT running, clear if they start running
IF (NOT IRC5Alarms[E_IRC5.AllTasksNotRunning].bRaised) AND (NOT ControllerIO.IN.AllTasksRunning) THEN
    IRC5Alarms[E_IRC5.AllTasksNotRunning].Raise(0);
ELSIF IRC5Alarms[E_IRC5.AllTasksNotRunning].bRaised AND (ControllerIO.IN.AllTasksRunning) THEN
    IRC5Alarms[E_IRC5.AllTasksNotRunning].Clear(0, 0);
END_IF;

///////////////////////////////////////////////////////////////////////////////
// 12. RunChainOK: ID=12
///////////////////////////////////////////////////////////////////////////////
IF (NOT IRC5Alarms[E_IRC5.RunChainOK].bRaised) AND (ControllerIO.IN.RunChainOK) THEN
    IRC5Alarms[E_IRC5.RunChainOK].Raise(0);
ELSIF IRC5Alarms[E_IRC5.RunChainOK].bRaised AND (NOT ControllerIO.IN.RunChainOK) THEN
    IRC5Alarms[E_IRC5.RunChainOK].Clear(0, 0);
END_IF;

///////////////////////////////////////////////////////////////////////////////
// 13. RunChainNotOK: ID=13
///////////////////////////////////////////////////////////////////////////////
IF (NOT IRC5Alarms[E_IRC5.RunChainNotOK].bRaised) AND (NOT ControllerIO.IN.RunChainOK) THEN
    IRC5Alarms[E_IRC5.RunChainNotOK].Raise(0);
ELSIF IRC5Alarms[E_IRC5.RunChainNotOK].bRaised AND (ControllerIO.IN.RunChainOK) THEN
    IRC5Alarms[E_IRC5.RunChainNotOK].Clear(0, 0);
END_IF;

///////////////////////////////////////////////////////////////////////////////
// 14. PP_Moved: ID=14
///////////////////////////////////////////////////////////////////////////////
IF (NOT IRC5Alarms[E_IRC5.PP_Moved].bRaised) AND (ControllerIO.IN.PP_Moved) THEN
    IRC5Alarms[E_IRC5.PP_Moved].Raise(0);
ELSIF IRC5Alarms[E_IRC5.PP_Moved].bRaised AND (NOT ControllerIO.IN.PP_Moved) THEN
    IRC5Alarms[E_IRC5.PP_Moved].Clear(0, 0);
END_IF;

// run the base extended monitoring
SUPER^.Monitoring();

//////////////////////////////////////////////////////////////////////////
// Wrap-up: Evaluate overall severity, after the extended Monitoring has ran base monitoring
//////////////////////////////////////////////////////////////////////////
_CurrentAlarmSeverity := F_GetMaxSeverityRaised(Alarms := IRC5Alarms, CurrentSeverity := _CurrentAlarmSeverity);
END_METHOD

METHOD SignalMapping : bool
VAR
END_VAR
OutputArray[0].0 := ControllerIO.OUT.PPtoMain;
OutputArray[0].1 := ControllerIO.OUT.Resume;
OutputArray[0].2 := ControllerIO.OUT.Pause;
OutputArray[0].3 := ControllerIO.OUT.EStopReset;
OutputArray[0].4 := ControllerIO.OUT.MotorsOn;
OutputArray[0].5 := ControllerIO.OUT.MotorsOff;

ControllerIO.IN.AutoMode          := InputArray[0].0;
ControllerIO.IN.E_Stop            := InputArray[0].1;
ControllerIO.IN.MotionSupervision := InputArray[0].2;
ControllerIO.IN.MotorsOn          := InputArray[0].3;
ControllerIO.IN.RunChainOK        := InputArray[0].4;
ControllerIO.IN.SignalsSimulated  := InputArray[0].5;
ControllerIO.IN.AllTasksRunning   := InputArray[0].6;
ControllerIO.IN.PP_Moved          := InputArray[0].7;
END_METHOD

METHOD Start : BOOL
VAR_INPUT
END_VAR
IF ControllerIO.IN.AllTasksRunning OR _Simulate THEN
    Start := TRUE;
    RETURN;
END_IF

Start := FALSE;

CASE _Start_State OF
    0:
        IF ControllerIO.IN.AllTasksRunning THEN
            _Start_State := 7;
        ELSE
            _Start_State := 1;
        END_IF

    1:
        ControllerIO.OUT.Resume := FALSE;
        ControllerIO.OUT.Pause  := FALSE;

        IF NOT ControllerIO.IN.E_Stop THEN
            _Start_State := 2;
        ELSIF ControllerIO.IN.RunChainOK THEN
            _Start_State := 3;
        END_IF

    2:
        ControllerIO.OUT.EStopReset := Pulse.PulseOutput;

        IF ControllerIO.IN.E_Stop = TRUE THEN
            ControllerIO.OUT.EStopReset := FALSE;
            _Start_State                := 1;
        END_IF

    3:
        IF ControllerIO.IN.AutoMode THEN
            _Start_State := 4;
        END_IF

    4:
        IF ControllerIO.IN.SignalsSimulated = TRUE THEN
            _Start_State := 5;
        END_IF

    5:
        ControllerIO.OUT.Resume := Pulse.PulseOutput;

        IF ControllerIO.IN.AllTasksRunning THEN
            ControllerIO.OUT.Resume := FALSE;
            _Start_State            := 7;
        ELSIF NOT ControllerIO.IN.RunChainOK THEN
            ControllerIO.OUT.Resume := FALSE;
            _Start_State            := 1;
        END_IF

    7:
        Start        := TRUE;
        _Start_State := 0;
END_CASE
END_METHOD

METHOD Stop : BOOL
VAR_INPUT
END_VAR
Stop := FALSE;

ControllerIO.OUT.Pause := ControllerIO.IN.AllTasksRunning;

IF NOT ControllerIO.IN.AllTasksRunning THEN
    ControllerIO.OUT.Pause := FALSE;
    Stop                   := TRUE;
END_IF
END_METHOD

PROPERTY EStopped : BOOL
GET
EStopped := NOT ControllerIO.IN.E_Stop;
END_GET
END_PROPERTY

PROPERTY InAuto : BOOL
GET
InAuto := ControllerIO.IN.AutoMode;
END_GET
END_PROPERTY

PROPERTY ParentResponseDefinitions : ARRAY[0..4] OF E_AlarmResponse
GET
IF _Simulate THEN
    ParentResponseDefinitions[TcEventSeverity.Verbose]  := E_AlarmResponse.NoResponse;
    ParentResponseDefinitions[TcEventSeverity.Info]     := E_AlarmResponse.NoResponse;
    ParentResponseDefinitions[TcEventSeverity.Warning]  := E_AlarmResponse.NoResponse;
    ParentResponseDefinitions[TcEventSeverity.Error]    := E_AlarmResponse.NoResponse;
    ParentResponseDefinitions[TcEventSeverity.Critical] := E_AlarmResponse.Suspend_Immediate;
ELSE
    ParentResponseDefinitions[TcEventSeverity.Verbose]  := E_AlarmResponse.NoResponse;
    ParentResponseDefinitions[TcEventSeverity.Info]     := E_AlarmResponse.NoResponse;
    ParentResponseDefinitions[TcEventSeverity.Warning]  := E_AlarmResponse.Suspend_Controlled;
    ParentResponseDefinitions[TcEventSeverity.Error]    := E_AlarmResponse.Suspend_Controlled;
    ParentResponseDefinitions[TcEventSeverity.Critical] := E_AlarmResponse.Suspend_Immediate;
END_IF
END_GET
END_PROPERTY

END_FUNCTION_BLOCK

// Machine/Components/MGB_Door/FB_Component_MGB_Door
FUNCTION_BLOCK FB_Component_MGB_Door EXTENDS FB_ComponentBase_SR
VAR_INPUT
    // Inputs

    EstopOK_CH1    : FB_DigitalSensor;
    EstopOK_CH2    : FB_DigitalSensor;
    AutoStopOK_CH1 : FB_DigitalSensor;
    AutoStopOK_CH2 : FB_DigitalSensor;
    Closed         : FB_DigitalSensor;
    mgbError       : FB_DigitalSensor;
    Pause          : FB_DigitalSensor;
    Resume         : FB_DigitalSensor;

    // Outputs
    Lock_Door  : FB_Component_Indicator;
    Reset_Door : FB_Component_Indicator;
    Estop_LED  : FB_Component_Indicator;
    Pause_LED  : FB_Component_Indicator;
    Resume_LED : FB_Component_Indicator;
END_VAR

VAR

    // Alarms
    StackLightAlarms : ARRAY[1..STACKLIGHT_ALARMS_COUNT] OF FB_TcAlarm;

    IsGreenFlashing : BOOL;
    IsRedFlashing   : BOOL;
    IsAmberFlashing : BOOL;
    HMI_DoorStatus  : ST_MGBDoor_HMIStatus;
    _SafetyReset    : BOOL;
    Sim_CloseDoor   : BOOL;
    Sim_ResetEstop  : BOOL;

    Sim_Reset_R_TRIG : R_TRIG;

END_VAR

VAR
    // Internal state variables
    DoorLocked   : BOOL := FALSE;
    PauseActive  : BOOL := FALSE;
    ResumeActive : BOOL := FALSE;
    EstopActive  : BOOL := FALSE;
END_VAR

VAR CONSTANT
    STACKLIGHT_ALARMS_COUNT : UDINT := 5;
END_VAR

//! @summary This method serves as the entry point for all underlying FB logic
METHOD PUBLIC CyclicLogic

//! @description This method should be called cyclically by descendant function blocks by invoking <c>SUPER^.CyclicLogic()</c>.  Alternatively, the contents of this method could be reimplemented entirely in which case a call to this method would not be necessary.
// Initialise Component
IF NOT _InitComplete THEN
    _InitComplete := Initialize();
    RETURN;
END_IF

EstopOK_CH1.CyclicLogic();
EstopOK_CH2.CyclicLogic();
AutoStopOK_CH1.CyclicLogic();
AutoStopOK_CH2.CyclicLogic();
Closed.CyclicLogic();
mgbError.CyclicLogic();
Pause.CyclicLogic();
Resume.CyclicLogic();

Lock_Door.CyclicLogic();
Pause_LED.CyclicLogic();
Resume_LED.CyclicLogic();
Estop_LED.CyclicLogic();

HMI_Status();

EstopOK_CH1.InSimulation    := _Simulate;
EstopOK_CH2.InSimulation    := _Simulate;
AutoStopOK_CH1.InSimulation := _Simulate;
AutoStopOK_CH2.InSimulation := _Simulate;

Sim_Reset_R_TRIG(CLK := _Simulate);

IF Sim_Reset_R_TRIG.Q THEN
    Sim_CloseDoor  := TRUE;
    Sim_ResetEstop := TRUE;
END_IF

IF Sim_CloseDoor THEN
    AutoStopOK_CH1.SimulationInput := TRUE;
    AutoStopOK_CH2.SimulationInput := TRUE;
ELSE
    AutoStopOK_CH1.SimulationInput := FALSE;
    AutoStopOK_CH2.SimulationInput := FALSE;
END_IF

IF Sim_ResetEstop THEN
    EstopOK_CH1.SimulationInput := TRUE;
    EstopOK_CH2.SimulationInput := TRUE;
ELSE
    EstopOK_CH1.SimulationInput := FALSE;
    EstopOK_CH2.SimulationInput := FALSE;
END_IF

// Call Super
SUPER^.CyclicLogic();

// Set Current Alarm Severity

////_CurrentAlarmSeverity := F_GetMaxSeverityRaised(Alarms := StackLightAlarms, CurrentSeverity := _CurrentSeverity, Severity := _CurrentAlarmSeverity);
END_METHOD

METHOD HMI_Status
VAR_INPUT
END_VAR

VAR_INST
    EStop_R_TRIG    : R_TRIG;
    AutoStop_R_TRIG : R_TRIG;
    EstopPressed    : BOOL;
    DoorOpened      : BOOL;
END_VAR
EStop_R_TRIG(CLK := NOT (EstopOK_CH1.Active AND EstopOK_CH2.Active));

IF EStop_R_TRIG.Q THEN
    EstopPressed := TRUE;
END_IF

IF _SafetyReset THEN
	EstopPressed := FALSE;
END_IF

HMI_DoorStatus.DoorName := Name;

IF EstopPressed THEN
    IF EstopOK_CH1.Active AND EstopOK_CH2.Active THEN
        HMI_DoorStatus.EStopStatus_Usint := 4;
        HMI_DoorStatus.EStopStatus_Str   := 'Reset Needed';
    ELSE
        HMI_DoorStatus.EStopStatus_Usint := 2;
        HMI_DoorStatus.EStopStatus_Str   := 'Estop Pressed';
    END_IF
ELSE
    IF EstopOK_CH1.Active AND EstopOK_CH2.Active THEN
        HMI_DoorStatus.EStopStatus_Usint := 1;
        HMI_DoorStatus.EStopStatus_Str   := 'Estop OK';
    ELSE
        HMI_DoorStatus.EStopStatus_Usint := 2;
        HMI_DoorStatus.EStopStatus_Str   := 'Estop Pressed';
    END_IF
END_IF

IF AutoStopOK_CH1.Active AND AutoStopOK_CH2.Active THEN
    HMI_DoorStatus.AutoStopStatus_Usint := 1;
    HMI_DoorStatus.AutoStopStatus_Str   := 'Door Closed';
ELSE
    HMI_DoorStatus.AutoStopStatus_Usint := 2;
    HMI_DoorStatus.AutoStopStatus_Str   := 'Door Open';
END_IF
END_METHOD

//! @summary Basic component initialization logic
METHOD PROTECTED Initialize : BOOL;

//! @description This method is called by <c>CyclicLogic()</c> as required
CreateEvents();

IF SUPER^.Initialize() THEN
    Initialize := TRUE;
END_IF
END_METHOD

PROPERTY AutoStop_CH_OK : BOOL
GET
AutoStop_CH_OK := AutoStopOK_CH1.Active AND AutoStopOK_CH2.Active;
END_GET
END_PROPERTY

PROPERTY Estop_CH_OK : BOOL
GET
Estop_CH_OK := EstopOK_CH2.Active AND EstopOK_CH1.Active;
END_GET
END_PROPERTY

PROPERTY SafetyReset : BOOL
SET
_SafetyReset := SafetyReset;
END_SET
END_PROPERTY

END_FUNCTION_BLOCK

// Machine/Components/Preplate_Rack/FB_Component_Preplate_Rack
FUNCTION_BLOCK FB_Component_Preplate_Rack EXTENDS FB_ComponentBase_SR
VAR_INPUT
    Executing : BOOL;

END_VAR

VAR
    // Inputs

    Button  : FB_Component_Button;
    Closed  : FB_DigitalSensor;
    _InAuto : BOOL;

    // Outputs
    Lock : FB_Component_Indicator;
END_VAR

VAR
    State    : E_RackState;
    R_Button : R_TRIG;

    //Properties
    _Available   : BOOL;
    _LinkBlocked : BOOL;
    _Blocked     : BOOL;
    Linked       : BOOL := TRUE;

    // Alarms
    RackDoorAlarms : ARRAY[1..RACK_DOOR_ALARMS_COUNT] OF FB_TcAlarm;

END_VAR

VAR
    // Internal state variables
    DoorLocked : BOOL := FALSE;
END_VAR

VAR CONSTANT
    RACK_DOOR_ALARMS_COUNT : UDINT := 5;
END_VAR

//! @summary This method serves as the entry point for all underlying FB logic
METHOD PUBLIC CyclicLogic

//! @description This method should be called cyclically by descendant function blocks by invoking <c>SUPER^.CyclicLogic()</c>.  Alternatively, the contents of this method could be reimplemented entirely in which case a call to this method would not be necessary.
RackLogic();

Button.CyclicLogic();
Closed.CyclicLogic();
Lock.CyclicLogic();

SUPER^.CyclicLogic();
END_METHOD

METHOD Block
VAR_INPUT
    Blocked : BOOL;
END_VAR
_Blocked := Blocked;
END_METHOD

METHOD Disable
VAR_INPUT
END_VAR
_Available := FALSE;
END_METHOD

//! @summary Basic component initialization logic
METHOD PROTECTED Initialize : BOOL;

//! @description This method is called by <c>CyclicLogic()</c> as required
CreateEvents();

IF SUPER^.Initialize() THEN
    Initialize := TRUE;
END_IF
END_METHOD

METHOD IsAvailable : BOOL
VAR_INPUT
END_VAR
IsAvailable := _Available;
END_METHOD

METHOD RackLogic
VAR_INPUT
END_VAR
R_Button(CLK := (Button.Button.Active));

CASE State OF
    E_RackState.Idle:
        Button.LED.TurnOn();
        Lock.TurnOn();
        _Available := TRUE;
        IF R_Button.Q THEN
            State := E_RackState.CheckForBlock;
        END_IF;

    E_RackState.CheckForBlock:
        Button.LED.Flash();
        Lock.TurnOn();
        IF NOT Blocked THEN
            State := E_RackState.CheckForLinked;
        ELSIF R_Button.Q THEN
            State := E_RackState.LockDoor;
        END_IF;

    E_RackState.CheckForLinked:
        Button.LED.Flash();
        IF NOT LinkBlocked THEN
            State := E_RackState.UnlockDoor;
        END_IF;

        IF NOT Linked THEN
            State := E_RackState.UnlockDoor;
        ELSIF R_Button.Q THEN
            State := E_RackState.LockDoor;
        END_IF;

    E_RackState.UnlockDoor:
        Lock.TurnOff();
        Button.LED.Flash();
        _Available := FALSE;
        State      := E_RackState.WaitForOpen;

    E_RackState.WaitForOpen:
        Button.LED.TurnOff();
        IF NOT Closed.Active THEN
            State := E_RackState.WaitForClose;
        END_IF;

    E_RackState.WaitForClose:
        Button.LED.TurnOff();
        IF Closed.Active THEN
            State := E_RackState.LockDoor;
        END_IF;

    E_RackState.LockDoor:
        Lock.TurnOn();
        Button.LED.Flash();
        State := E_RackState.EnableDoor;

    E_RackState.EnableDoor:
        Lock.TurnOn();
        _Available := TRUE;
        State      := E_RackState.Idle;
END_CASE;

IF NOT Executing THEN
    Lock.TurnOff();

END_IF
END_METHOD

PROPERTY Blocked : BOOL
GET
Blocked := _Blocked;
END_GET
SET
_Blocked := Blocked;
END_SET
END_PROPERTY

PROPERTY PUBLIC InAuto : BOOL
SET
_InAuto := InAuto;
END_SET
END_PROPERTY

PROPERTY LinkBlocked : BOOL
GET
LinkBlocked := _LinkBlocked;
END_GET
SET
_LinkBlocked := LinkBlocked;
END_SET
END_PROPERTY

END_FUNCTION_BLOCK

// Machine/Components/Robot/FB_Component_Robot
FUNCTION_BLOCK FB_Component_Robot EXTENDS FB_ComponentBase_SR
VAR_INPUT
    Handshake         : ST_Robot_Handshake_IO;
    RecipeData_ToSend : ARRAY[0..14] OF DINT;
    Current_StepNum   : UINT;

END_VAR

VAR
    Robot_Name : STRING;

    InputArray       AT %I* : ARRAY[0..7] OF USINT;
    OtherInputsArray AT %I* : ARRAY[0..7] OF USINT;

    // Outputs
    OutputArray       AT %Q* : ARRAY[0..7] OF USINT;
    OtherOutputsArray AT %Q* : ARRAY[0..7] OF USINT;

    Recipe_PackedBytes AT %Q* : ARRAY[0..16] OF USINT; // Maximum size of packed bytes array
    Recipe_ByteQtyKey  AT %Q* : ARRAY[0..14] OF USINT; // Array to store the number of bytes for each number

END_VAR

//! @summary This method serves as the entry point for all underlying FB logic
METHOD PUBLIC CyclicLogic

//! @description This method should be called cyclically by descendant function blocks by invoking <c>SUPER^.CyclicLogic()</c>.  Alternatively, the contents of this method could be reimplemented entirely in which case a call to this method would not be necessary.
// Initialise Component

IF NOT _InitComplete THEN
    _InitComplete := Initialize();
    RETURN;
END_IF

// map signals
HandshakeSignalMapping();

PackRecipeData();

// Call Super

SUPER^.CyclicLogic();

// Set Current Alarm Severity

_CurrentAlarmSeverity := F_GetMaxSeverityRaised(Alarms := Comp_Alarms, CurrentSeverity := _CurrentAlarmSeverity);
END_METHOD

METHOD Clear_DataToSend : BOOL
VAR_INPUT
END_VAR
FOR i := 0 TO 14 DO
    RecipeData_ToSend[i] := 0;
END_FOR
END_METHOD

METHOD PROTECTED CreateEvents
VAR_INPUT
END_VAR
SUPER^.CreateEvents();
END_METHOD

METHOD HandshakeSignalMapping : bool
VAR
END_VAR
OutputArray[0].0 := Handshake.OUT.Execute_Step;
OutputArray[0].1 := Handshake.OUT.MessageAcknowledge;
OutputArray[0].2 := Handshake.OUT.Execute_Service;

memcpy(ADR(OutputArray[2]), ADR(Handshake.OUT.Execute_StepNum), 2);

//SubStepNumber is an enumerator and that is a DINT and we need it to only be a USINT
memcpy(ADR(OutputArray[4]), ADR(Handshake.OUT.SubStepResponse), 1);

//	OutputArray[4] := Handshake.OUT.SubStepResponse;
OutputArray[5] := Handshake.OUT.MessageSolution;
OutputArray[6] := Handshake.OUT.Execute_ServiceNum;

Handshake.IN.Executing_Step    := InputArray[0].0;
Handshake.IN.StepComplete      := InputArray[0].1;
Handshake.IN.ErrorPresent      := InputArray[0].2;
Handshake.IN.Executing_Service := InputArray[0].3;
Handshake.IN.ServiceComplete   := InputArray[0].4;
Handshake.IN.TaskRunning       := InputArray[0].5;

memcpy(ADR(Handshake.IN.MessageNumber), ADR(InputArray[2]), 2);

//SubStepNumber is an enumerator and that is a DINT and we need it to only be a USINT
memcpy(ADR(Handshake.IN.SubStepNumber), ADR(InputArray[4]), 1);
END_METHOD

//! @summary Basic component initialization logic
METHOD PROTECTED Initialize : BOOL;

//! @description This method is called by <c>CyclicLogic()</c> as required
CreateEvents();

IF SUPER^.Initialize() THEN
    Initialize := TRUE;
END_IF
END_METHOD

METHOD PROTECTED Monitoring
VAR_INPUT
END_VAR
SUPER^.Monitoring();
END_METHOD

METHOD PackRecipeData : BOOL
VAR
    i, j         : INT; // Loop counters
    index        : INT; // Temporary variable to hold the number
    numberToPack : UDINT;
END_VAR
// The Bitmask range for each robot (32 bytes) is divided into two sections, one for key values and one for data

// The key section includes 15 bytes, one for each possible data field

